(* IEC 61131-3 sources: std_i2980_v2.06_cp053/Source/IMM/ieccontrol/PumpGeneral (part 2) *)

(* ---- ABPumpOutput.pu ---- *)
(*
@h    ! WARNING !
@h    The Kemro K2 system (including software) only meets category B according to EN 954-1,
@h    thus it is not intended for usage in safety-relevant control applications in the field
@h    of personal safety (e.g. emergency stop).
@h    To implement potentially necessary safety-relevant control tasks, always use additional
@h    external safety devices that are intended for the particular purpose, and meet the necessary
@h    functional safety.
@h    For further information see EN 954-1 (EN ISO 13849-1) and/or the K2-x00 user manual, chapter
@h    "CE conformity, directives and standards".

This AB starts and stopps the process algorithms for fast output and mid output.
After a change in pressure or velocity lintab, a minimum output voltage is calculated.
During operation modes manual, HA and FA the output to the pump is at least this calculated minimum voltage,
even if there is actually no movement active.
In setup mode, the output voltage is set to 0.0 if the pump is stopped.
This block offers also the possibility to add a dither signal to pressure and velocity output.
Setting the dither amplitude to 0.0 disables the signal.
If the application is not running on a CP 03x, the dither amplitude is automatically resetted to 0.0.
*)

IMPORT_OVER_LISTFILE
 SET_ALARM
, GET_SYNC_REFTO
, WRITE_SVREAL_DIRECT
, FAddToScopeGroup
, ABAnalogOutput
, ABAnalogHWOut
, tsDeviceId
, KAPPL_LintabData
, tnOperationMode
, tnAnaOutputMode
, FBDebugTrace
, FBSinus
, KSWO_Status
, KCTRL_Lintab_Light
, KCTRL_Lintab_Param_Light
, KCAT_HandleData
, KCAT_Status

END_IMPORT

ALGORITHM_BLOCK ABPumpOutput #DUMMY_EDIT_BLOCK

SYSTEM_VAR
 sv_rPressure : REAL;
 sv_rVelocity : REAL;
 sv_DeviceId : tsDeviceId;
 sv_rMinVoltageVelOutput : REAL;
 sv_rMinVoltagePressOutput : REAL;
 sv_VelocityLintab : KAPPL_LintabData;
 sv_PressureLintab : KAPPL_LintabData;
 sv_OperationMode : tnOperationMode;
 sv_rValueMinVoltageVelDetect : REAL (* x - value [%] for detection of minimum output voltage of AO pump velocity *);
 sv_rValueMinVoltagePresDetect : REAL (* x - value [bar] for detection of minimum output voltage of AO pump pressure *);
 sv_rDitherFrequencyVel : REAL;
 sv_rDitherAmplitudeVel : REAL;
 sv_rDitherFrequencyPres : REAL;
 sv_rDitherAmplitudePres : REAL;
 sv_bInitStart : BOOL;
 sv_bInitDone : BOOL;
 sv_rMaxPressure : REAL;
END_VAR

SYSTEM_OBJECT
 TaskAnalog : TASK;
 TaskInject : TASK;
 TaskSlow : TASK;
 erVariableNotLinked : ALARM;
 PU_Task_7 : TASK;
 PU_Task_3 : TASK;
END_OBJECT

VAR
 mbStop : BOOL;
 mbStopped : BOOL := TRUE;
 mprPressureSource : REFTO REAL;
 mprVelocitySource : REFTO REAL;
 abAnalogOutputP : ABAnalogOutput;
 abAnalogOutputV : ABAnalogOutput;
 abAnalogHWOutP : ABAnalogHWOut;
 abAnalogHWOutV : ABAnalogHWOut;
 mrMinVoltageVelocityOutput : REAL (* minimum voltage for AO velocity (only considered in HA and FA) *);
 mrMinVoltagePressureOutput : REAL (* minimum voltage for AO pressure (only considered in HA and FA) *);
END_VAR

ALGORITHM aStart

VAR_INPUT
 AnaOutMode : tnAnaOutputMode;
 pLintabP : REFTO KAPPL_LintabData;
 pLintabV : REFTO KAPPL_LintabData;
 prPressure : REFTO REAL;
 prVelocity : REFTO REAL;
END_VAR
#BEGIN_EDIT_BLOCK
(**************************************** WARNING ********************************************
 *** The KEBA Kemro K2 System including software is not intended for safety control tasks! ***
 ***                       For further information see Comment tab!                        ***
 *********************************************************************************************)

mbStop := FALSE;
//make sure when we get a start and a stop very fast,
//we do not end up in a situation where mbStopped is FALSE but paXxxOutput is still running
mbStopped := FALSE;

abAnalogOutputP.aInit(pLintab := pLintabP);
abAnalogOutputV.aInit(pLintab := pLintabV);

mprPressureSource := prPressure;
mprVelocitySource := prVelocity;

CASE AnaOutMode OF

   nAnaOutputModeMid:
         START_PROCESS_ALGORITHM(paMidOutput);

   nAnaOutputModeFast:
         START_PROCESS_ALGORITHM(paFastOutput);
END_CASE;

;#END_EDIT_BLOCK END_ALGORITHM

ALGORITHM aStop

VAR_OUTPUT
 bReady : BOOL;
END_VAR
#BEGIN_EDIT_BLOCK
(**************************************** WARNING ********************************************
 *** The KEBA Kemro K2 System including software is not intended for safety control tasks! ***
 ***                       For further information see Comment tab!                        ***
 *********************************************************************************************)

IF NOT mbStopped THEN
   mbStop := TRUE;
END_IF;
bReady := mbStopped;

;#END_EDIT_BLOCK END_ALGORITHM

ALGORITHM aSetErrorMessage

VAR
 fbDebugTrace : FBDebugTrace;
END_VAR
#BEGIN_EDIT_BLOCK
(**************************************** WARNING ********************************************
 *** The KEBA Kemro K2 System including software is not intended for safety control tasks! ***
 ***                       For further information see Comment tab!                        ***
 *********************************************************************************************)

IF NOT abAnalogHWOutV.aIsLinked() THEN
   SET_ALARM(Name := erVariableNotLinked,
             SubID1 := sv_DeviceId.CompId,
             SubID2 := sv_DeviceId.IndexId,
             Param1 := 'ao_Velocity');
END_IF;

IF NOT abAnalogHWOutP.aIsLinked() THEN
   SET_ALARM(Name := erVariableNotLinked,
             SubID1 := sv_DeviceId.CompId,
             SubID2 := sv_DeviceId.IndexId,
             Param1 := 'ao_Pressure');
END_IF;

IF abAnalogOutputP.aRun.bError THEN
   fbDebugTrace(CONCAT('ABPumpOutput: error ',DINT_TO_STRING(abAnalogOutputP.aRun.iErrorInfo),' in ABAnalogOutputP'));
END_IF;

IF abAnalogOutputV.aRun.bError THEN
   fbDebugTrace(CONCAT('ABPumpOutput: error ',DINT_TO_STRING(abAnalogOutputV.aRun.iErrorInfo),' in ABAnalogOutputV'));
END_IF;

;#END_EDIT_BLOCK END_ALGORITHM

PROCESS_ALGORITHM paFastOutput ON TaskInject(15000)

VAR_TEMP
 b : BOOL;
END_VAR

VAR
 fbSinusVel : FBSinus;
 fbSinusPres : FBSinus;
 rDitherVel : REAL;
 rDitherPres : REAL;
 rPressure : REAL;
END_VAR

(* IecGraph-Code *)

(* init step *)
INITIAL_STEP OUT:
Init (P);
ADitherSignal (N);
AOUT (N);
END_STEP

ACTION Init: #BEGIN_EDIT_BLOCK
mbStopped := FALSE;

;#END_EDIT_BLOCK END_ACTION (*Init*)
ACTION AOUT: #BEGIN_EDIT_BLOCK
//limit pressure output to max. pressure of the pump
rPressure := MIN(sv_rMaxPressure, mprPressureSource^);

b := WRITE_SVREAL_DIRECT(sv_rPressure, rPressure);
b := WRITE_SVREAL_DIRECT(sv_rVelocity, mprVelocitySource^);

(* Lintab Calculation *)
abAnalogOutputP.aRun(rSetValue := sv_rPressure);
abAnalogOutputV.aRun(rSetValue := sv_rVelocity);

(* Output to AO and Shortcircuit detection *)
abAnalogHWOutP.aOut(rValue := (MAX(abAnalogOutputP.aRun.rOutput, mrMinVoltagePressureOutput)) + rDitherPres);
abAnalogHWOutV.aOut(rValue := (MAX(abAnalogOutputV.aRun.rOutput, mrMinVoltageVelocityOutput)) + rDitherVel);

;#END_EDIT_BLOCK END_ACTION (*AOUT*)

(* steps *)
STEP ERROR_STOP:
AErrorStop (P);
END_STEP

ACTION AErrorStop: #BEGIN_EDIT_BLOCK
sv_rPressure := 0.0;
sv_rVelocity := 0.0;
aSetErrorMessage();

;#END_EDIT_BLOCK END_ACTION (*AErrorStop*)
STEP S_Stop:
AStop (P);
END_STEP

ACTION AStop: #BEGIN_EDIT_BLOCK
mbStop := FALSE;

(* Stopping Analog Output*)
abAnalogHWOutP.aOut(rValue := mrMinVoltagePressureOutput);
abAnalogHWOutV.aOut(rValue := mrMinVoltageVelocityOutput);

mbStopped := TRUE;
STOP_PROCESS_ALGORITHM();

;#END_EDIT_BLOCK END_ACTION (*AStop*)

(* transitions *)
TRANSITION Trans1 (* Trans1 *) FROM OUT TO ERROR_STOP :=  #BEGIN_EDIT_BLOCK
abAnalogOutputP.aRun.bError OR
abAnalogOutputV.aRun.bError OR
abAnalogHWOutP.aOut.bError OR
abAnalogHWOutV.aOut.bError
;#END_EDIT_BLOCK
END_TRANSITION

GO_ON_TRANSITION Trans5 (* Trans5 *) FROM ERROR_STOP TO S_Stop :=  #BEGIN_EDIT_BLOCK
TRUE
;#END_EDIT_BLOCK
END_TRANSITION

GO_ON_TRANSITION TStop (* Trans4 *) FROM OUT TO S_Stop :=  #BEGIN_EDIT_BLOCK
mbStop
;#END_EDIT_BLOCK
END_TRANSITION

TRANSITION TNewOutput (* Trans7 *) FROM S_Stop TO OUT :=  #BEGIN_EDIT_BLOCK
TRUE
;#END_EDIT_BLOCK
END_TRANSITION

(* end IecGraph-Code *)
(* sfc-code *)

(* stand alone actions *)
ACTION ADitherSignal: #BEGIN_EDIT_BLOCK
(**************************************** WARNING ********************************************
 *** The KEBA Kemro K2 System including software is not intended for safety control tasks! ***
 ***                       For further information see Comment tab!                        ***
 *********************************************************************************************)

//sinus signals for pressure and velocity dither
IF sv_rDitherAmplitudeVel > 0.0 THEN
   fbSinusVel(rAmplitude := sv_rDitherAmplitudeVel,
              rFrequency := sv_rDitherFrequencyVel,
              rOut => rDitherVel);
ELSE
   rDitherVel := 0.0;
END_IF;

IF sv_rDitherAmplitudePres > 0.0 THEN
   fbSinusPres(rAmplitude := sv_rDitherAmplitudePres,
              rFrequency := sv_rDitherFrequencyPres,
              rOut => rDitherPres);
ELSE
   rDitherPres := 0.0;
END_IF;

;#END_EDIT_BLOCK END_ACTION (*ADitherSignal*)
(* end sfc-code *)

END_ALGORITHM

PROCESS_ALGORITHM paMidOutput ON TaskAnalog(15000)

VAR_TEMP
 b : BOOL;
END_VAR

VAR
 fbSinusVel : FBSinus;
 fbSinusPres : FBSinus;
 rDitherVel : REAL;
 rDitherPres : REAL;
 rPressure : REAL;
END_VAR

(* IecGraph-Code *)

(* init step *)
INITIAL_STEP OUT:
Init (P);
ADitherSignal (N);
AOUT (N);
END_STEP

ACTION Init: #BEGIN_EDIT_BLOCK
mbStopped := FALSE;

;#END_EDIT_BLOCK END_ACTION (*Init*)
ACTION AOUT: #BEGIN_EDIT_BLOCK
//limit pressure output to max. pressure of the pump
rPressure := MIN(sv_rMaxPressure, mprPressureSource^);

b := WRITE_SVREAL_DIRECT(sv_rPressure, rPressure);
b := WRITE_SVREAL_DIRECT(sv_rVelocity, mprVelocitySource^);

(* Lintab Calculation *)
abAnalogOutputP.aRun(rSetValue := sv_rPressure);
abAnalogOutputV.aRun(rSetValue := sv_rVelocity);

(* Shortcircuit detection *)
abAnalogHWOutP.aOut(rValue := (MAX(abAnalogOutputP.aRun.rOutput, mrMinVoltagePressureOutput)) + rDitherPres);
abAnalogHWOutV.aOut(rValue := (MAX(abAnalogOutputV.aRun.rOutput, mrMinVoltageVelocityOutput)) + rDitherVel);

;#END_EDIT_BLOCK END_ACTION (*AOUT*)

(* steps *)
STEP ERROR_STOP:
AErrorStop (P);
END_STEP

ACTION AErrorStop: #BEGIN_EDIT_BLOCK
sv_rPressure := 0.0;
sv_rVelocity := 0.0;
aSetErrorMessage();

;#END_EDIT_BLOCK END_ACTION (*AErrorStop*)
STEP S_Stop:
AStop (P);
END_STEP

ACTION AStop: #BEGIN_EDIT_BLOCK
mbStop := FALSE;

(* Stopping Analog Output*)
abAnalogHWOutP.aOut(rValue := mrMinVoltagePressureOutput);
abAnalogHWOutV.aOut(rValue := mrMinVoltageVelocityOutput);

mbStopped := TRUE;
STOP_PROCESS_ALGORITHM();

;#END_EDIT_BLOCK END_ACTION (*AStop*)

(* transitions *)
TRANSITION Trans1 (* Trans1 *) FROM OUT TO ERROR_STOP :=  #BEGIN_EDIT_BLOCK
abAnalogOutputP.aRun.bError OR
abAnalogOutputV.aRun.bError OR
abAnalogHWOutP.aOut.bError OR
abAnalogHWOutV.aOut.bError
;#END_EDIT_BLOCK
END_TRANSITION

GO_ON_TRANSITION Trans5 (* Trans5 *) FROM ERROR_STOP TO S_Stop :=  #BEGIN_EDIT_BLOCK
TRUE
;#END_EDIT_BLOCK
END_TRANSITION

GO_ON_TRANSITION TStop (* Trans4 *) FROM OUT TO S_Stop :=  #BEGIN_EDIT_BLOCK
mbStop
;#END_EDIT_BLOCK
END_TRANSITION

TRANSITION TNewOutput (* Trans7 *) FROM S_Stop TO OUT :=  #BEGIN_EDIT_BLOCK
TRUE
;#END_EDIT_BLOCK
END_TRANSITION

(* end IecGraph-Code *)
(* sfc-code *)

(* stand alone actions *)
ACTION ADitherSignal: #BEGIN_EDIT_BLOCK
(**************************************** WARNING ********************************************
 *** The KEBA Kemro K2 System including software is not intended for safety control tasks! ***
 ***                       For further information see Comment tab!                        ***
 *********************************************************************************************)

//sinus signals for pressure and velocity dither
IF sv_rDitherAmplitudeVel > 0.0 THEN
   fbSinusVel(rAmplitude := sv_rDitherAmplitudeVel,
              rFrequency := sv_rDitherFrequencyVel,
              rOut => rDitherVel);
ELSE
   rDitherVel := 0.0;
END_IF;

IF sv_rDitherAmplitudePres > 0.0 THEN
   fbSinusPres(rAmplitude := sv_rDitherAmplitudePres,
              rFrequency := sv_rDitherFrequencyPres,
              rOut => rDitherPres);
ELSE
   rDitherPres := 0.0;
END_IF;

;#END_EDIT_BLOCK END_ACTION (*ADitherSignal*)
(* end sfc-code *)

END_ALGORITHM

PROCESS_ALGORITHM paInitDebugMeasurement ON TaskSlow AUTOSTART

VAR
 fuName : STRING(255);
 variableName : STRING(255);
 swoState : KSWO_Status;
 b : BOOL;
END_VAR
#BEGIN_EDIT_BLOCK
fuName := GET_MY_FU_NAME();
variableName := CONCAT(fuName,'.rPressure Hydr bar');
swoState := KSWO_AddVariable( Task := TaskInject,
                              Name := variableName,
                              Variable := sv_rPressure);
b := FAddToScopeGroup(Task := TaskInject,
                      Name := variableName,
                      GroupId := cScopeGroupPump);
variableName := CONCAT(fuName,'.rVelocity %');
swoState := KSWO_AddVariable( Task := TaskInject,
                              Name := variableName,
                              Variable := sv_rVelocity);
b := FAddToScopeGroup(Task := TaskInject,
                      Name := variableName,
                      GroupId := cScopeGroupPump);

variableName := CONCAT(fuName,'.rPressure Hydr bar');
swoState := KSWO_AddVariable( Task := TaskAnalog,
                              Name := variableName,
                              Variable := sv_rPressure);
variableName := CONCAT(fuName,'.rVelocity %');
swoState := KSWO_AddVariable( Task := TaskAnalog,
                              Name := variableName,
                              Variable := sv_rVelocity);

STOP_PROCESS_ALGORITHM();

;#END_EDIT_BLOCK END_ALGORITHM

ALGORITHM aGetMinVoltage

VAR_INPUT
 pLintab : REFTO KAPPL_LintabData;
 rXValue : REAL (* xValue (for example 1% or 2 bar) *);
END_VAR

VAR_OUTPUT
 rMinVoltage : REAL (* according voltage for rXValue *);
END_VAR

VAR
 Lintab : KCTRL_Lintab_Light;
 LintabParams : KCTRL_Lintab_Param_Light;
END_VAR
#BEGIN_EDIT_BLOCK
(**************************************** WARNING ********************************************
 *** The KEBA Kemro K2 System including software is not intended for safety control tasks! ***
 ***                       For further information see Comment tab!                        ***
 *********************************************************************************************)

LintabParams.LintabPoints := pLintab^.LintabPoints;
LintabParams.Mode.bLinearExtrapolation := TRUE;
LintabParams.Mode.bSetNegativeValuesToZero := FALSE;
LintabParams.Mode.bZeroExtrapolation := FALSE;
Lintab.Par(Param := LintabParams);

IF Lintab.Par.parStatus <> KCTRL_Ret_OK THEN
   rMinVoltage := 0.0;
   RETURN; //error -> return 0.0
END_IF;

//calculate value
Lintab.Calculate(rX := rXValue);
IF Lintab.Calculate.calcStatus <> KCTRL_Ret_OK THEN
   rMinVoltage := 0.0;
   RETURN; //error -> return 0.0
ELSE
   rMinVoltage := Lintab.Calculate.rY;
END_IF;

;#END_EDIT_BLOCK END_ALGORITHM

POSTUPDATE_ALGORITHM pVelocityLintab ON PU_Task_7 WITH sv_VelocityLintab,sv_rValueMinVoltageVelDetect

#BEGIN_EDIT_BLOCK
(**************************************** WARNING ********************************************
 *** The KEBA Kemro K2 System including software is not intended for safety control tasks! ***
 ***                       For further information see Comment tab!                        ***
 *********************************************************************************************)

aGetMinVoltage(pLintab := @sv_VelocityLintab,
               rXValue := sv_rValueMinVoltageVelDetect,
               rMinVoltage => sv_rMinVoltageVelOutput);

;#END_EDIT_BLOCK END_ALGORITHM

POSTUPDATE_ALGORITHM pPressureLintab ON PU_Task_7 WITH sv_PressureLintab,sv_rValueMinVoltagePresDetect

#BEGIN_EDIT_BLOCK
(**************************************** WARNING ********************************************
 *** The KEBA Kemro K2 System including software is not intended for safety control tasks! ***
 ***                       For further information see Comment tab!                        ***
 *********************************************************************************************)

aGetMinVoltage(pLintab := @sv_PressureLintab,
               rXValue := sv_rValueMinVoltagePresDetect,
               rMinVoltage => sv_rMinVoltagePressOutput);

;#END_EDIT_BLOCK END_ALGORITHM

POSTUPDATE_ALGORITHM pDitherParams ON PU_Task_7 WITH sv_bInitStart,sv_rDitherAmplitudePres,sv_rDitherAmplitudeVel

VAR
 HandleData : KCAT_HandleData;
 CatStatus : KCAT_Status;
 sDevice : STRING(31);
 bInitDone : BOOL;
 bCurrentOutput : BOOL (* TRUE: current output available *);
END_VAR
#BEGIN_EDIT_BLOCK
(**************************************** WARNING ********************************************
 *** The KEBA Kemro K2 System including software is not intended for safety control tasks! ***
 ***                       For further information see Comment tab!                        ***
 *********************************************************************************************)

IF NOT bInitDone THEN
   //get device name
   HandleData := KCAT_GetHandle('IO.ONBOARD.deviceName');
   IF HandleData.Status = KCAT_Status_OK THEN
      CatStatus := KCAT_GetValue(Handle := HandleData.Handle, Buffer := sDevice);
      sDevice := LEFT(sDevice,5);

      IF sDevice ='CP 03' THEN
         bCurrentOutput := TRUE;
      END_IF;
   END_IF;

   bInitDone := TRUE;

END_IF;

IF NOT bCurrentOutput THEN
   //set dither amplitude to 0.0 (=disable dither signal)
   sv_rDitherAmplitudeVel := 0.0;
   sv_rDitherAmplitudePres := 0.0;
END_IF;

;#END_EDIT_BLOCK END_ALGORITHM

POSTUPDATE_ALGORITHM pSetMinVoltage ON PU_Task_3 WITH sv_bInitDone,sv_rMinVoltageVelOutput,sv_rMinVoltagePressOutput,sv_OperationMode

#BEGIN_EDIT_BLOCK
(**************************************** WARNING ********************************************
 *** The KEBA Kemro K2 System including software is not intended for safety control tasks! ***
 ***                       For further information see Comment tab!                        ***
 *********************************************************************************************)

IF sv_OperationMode = nSetup THEN
   //setup mode -> set minimum output voltage to 0.0
   mrMinVoltagePressureOutput := 0.0;
   mrMinVoltageVelocityOutput := 0.0;

ELSE
   //all other operation modes
   mrMinVoltagePressureOutput := sv_rMinVoltagePressOutput;
   mrMinVoltageVelocityOutput := sv_rMinVoltageVelOutput;
END_IF;

IF mbStopped THEN
   //write to AO´s immediately if device is not active
   abAnalogHWOutP.aOut(rValue := mrMinVoltagePressureOutput);
   abAnalogHWOutV.aOut(rValue := mrMinVoltageVelocityOutput);
END_IF;

;#END_EDIT_BLOCK END_ALGORITHM

END_ALGORITHM_BLOCK

#END_OF_IEC_PART

@Puma @IecEditor 6 97 @Pou 25
@@@BEG_Comment@@@
@h    ! WARNING !
@h    The Kemro K2 system (including software) only meets category B according to EN 954-1,
@h    thus it is not intended for usage in safety-relevant control applications in the field
@h    of personal safety (e.g. emergency stop).
@h    To implement potentially necessary safety-relevant control tasks, always use additional
@h    external safety devices that are intended for the particular purpose, and meet the necessary
@h    functional safety.
@h    For further information see EN 954-1 (EN ISO 13849-1) and/or the K2-x00 user manual, chapter
@h    "CE conformity, directives and standards".

This AB starts and stopps the process algorithms for fast output and mid output.
After a change in pressure or velocity lintab, a minimum output voltage is calculated.
During operation modes manual, HA and FA the output to the pump is at least this calculated minimum voltage,
even if there is actually no movement active.
In setup mode, the output voltage is set to 0.0 if the pump is stopped.
This block offers also the possibility to add a dither signal to pressure and velocity output.
Setting the dither amplitude to 0.0 disables the signal.
If the application is not running on a CP 03x, the dither amplitude is automatically resetted to 0.0.
@@@END_Comment@@@

@BEG_Contents

@BEG_Func
@RT(17)FuncTreeContainer
4
@Var @RT(9)SET_ALARM @RT(0) @T @T @DERIVED 0 @F @RT(23)KEBA_STANDARD_PROCEDURE @F
@T
@BEG_Attrib
0 @RT(0) @RT(0)
@END_Attrib
1 1 @F @F @F @F

@Var @RT(14)GET_SYNC_REFTO @RT(0) @T @T @DERIVED 0 @F @RT(22)KEBA_STANDARD_FUNCTION @F
@T
@BEG_Attrib
0 @RT(0) @RT(0)
@END_Attrib
1 1 @F @F @F @F

@Var @RT(19)WRITE_SVREAL_DIRECT @RT(0) @T @T @DERIVED 0 @F @RT(22)KEBA_STANDARD_FUNCTION @F
@T
@BEG_Attrib
0 @RT(0) @RT(0)
@END_Attrib
1 1 @F @F @F @F

@Var @RT(16)FAddToScopeGroup @RT(0) @T @T @DERIVED 0 @F @RT(8)FUNCTION @F
@T
@BEG_Attrib
0 @RT(0) @RT(0)
@END_Attrib
1 1 @F @F @F @F

@END_Func

@BEG_Const
@RT(18)ConstTreeContainer
0
@END_Const

@BEG_Export

@BEG_Kind
@ALGORITHM_BLOCK @RT(12)ABPumpOutput @STRUCTURED_TEXT
@RT(0) @RT(0) @RT(0)
@END_Kind

@BEG_Dcl
@RT(16)DclTreeContainer
33
@Var @RT(10)TaskAnalog @RT(0) @T @T @RENAMED 0 @T @T @DT @RT(4)TASK @RT(0) @T @T @BASIC 0 @F
@F @F
@T
@BEG_Attrib
3 @RT(0) @RT(0) @RT(0)
@END_Attrib
1 7 @F @F @F @F

@Var @RT(10)TaskInject @RT(0) @T @T @RENAMED 0 @T @T @DT @RT(4)TASK @RT(0) @T @T @BASIC 0 @F
@F @F
@T
@BEG_Attrib
3 @RT(0) @RT(0) @RT(0)
@END_Attrib
1 7 @F @F @F @F

@Var @RT(8)TaskSlow @RT(0) @T @T @RENAMED 0 @T @T @DT @RT(4)TASK @RT(0) @T @T @BASIC 0 @F
@F @F
@T
@BEG_Attrib
3 @RT(0) @RT(0) @RT(0)
@END_Attrib
1 7 @F @F @F @F

@Var @RT(12)sv_rPressure @RT(0) @T @F @DT @RT(4)REAL @RT(0) @T @T @BASIC 0 @F
@F @F
@T
@BEG_Attrib
3 @RT(0) @RT(0) @RT(0)
@END_Attrib
1 8 @F @F @F @F

@Var @RT(12)sv_rVelocity @RT(0) @T @F @DT @RT(4)REAL @RT(0) @T @T @BASIC 0 @F
@F @F
@T
@BEG_Attrib
3 @RT(0) @RT(0) @RT(0)
@END_Attrib
1 8 @F @F @F @F

@Var @RT(6)mbStop @RT(0) @T @F @DT @RT(4)BOOL @RT(0) @T @T @BASIC 0 @F
@F @F
@T
@BEG_Attrib
3 @RT(0) @RT(0) @RT(0)
@END_Attrib
1 0 @F @F @F @F

@Var @RT(9)mbStopped @RT(0) @T @F @DT @RT(4)BOOL @RT(0) @T @T @BASIC 0 @F
@F @F
@T
@BEG_Attrib
3 @RT(4)TRUE @RT(0) @RT(0)
@END_Attrib
1 0 @F @F @F @F

@Var @RT(17)mprPressureSource @RT(0) @T @T @REFTO 0 @T @DT @RT(4)REAL @RT(0) @T @T @BASIC 0 @F
@F @F
@T
@BEG_Attrib
3 @RT(0) @RT(0) @RT(0)
@END_Attrib
1 0 @F @F @F @F

@Var @RT(17)mprVelocitySource @RT(0) @T @T @REFTO 0 @T @DT @RT(4)REAL @RT(0) @T @T @BASIC 0 @F
@F @F
@T
@BEG_Attrib
3 @RT(0) @RT(0) @RT(0)
@END_Attrib
1 0 @F @F @F @F

@Var @RT(15)abAnalogOutputP @RT(0) @T @T @DERIVED 0 @T @T @DT @RT(14)ABAnalogOutput @RT(0) @T @T @UNKNOWN 0 @F
@F @F
@T
@BEG_Attrib
3 @RT(0) @RT(0) @RT(0)
@END_Attrib
1 0 @F @F @F @F

@Var @RT(15)abAnalogOutputV @RT(0) @T @T @DERIVED 0 @T @T @DT @RT(14)ABAnalogOutput @RT(0) @T @T @UNKNOWN 0 @F
@F @F
@T
@BEG_Attrib
3 @RT(0) @RT(0) @RT(0)
@END_Attrib
1 0 @F @F @F @F

@Var @RT(14)abAnalogHWOutP @RT(0) @T @T @DERIVED 0 @T @T @DT @RT(13)ABAnalogHWOut @RT(0) @T @T @UNKNOWN 0 @F
@F @F
@T
@BEG_Attrib
3 @RT(0) @RT(0) @RT(0)
@END_Attrib
1 0 @F @F @F @F

@Var @RT(14)abAnalogHWOutV @RT(0) @T @T @DERIVED 0 @T @T @DT @RT(13)ABAnalogHWOut @RT(0) @T @T @UNKNOWN 0 @F
@F @F
@T
@BEG_Attrib
3 @RT(0) @RT(0) @RT(0)
@END_Attrib
1 0 @F @F @F @F

@Var @RT(19)erVariableNotLinked @RT(0) @T @F @DT @RT(5)ALARM @RT(0) @T @T @BASIC 0 @F
@F @F
@T
@BEG_Attrib
3 @RT(0) @RT(0) @RT(0)
@END_Attrib
1 7 @F @F @F @F

@Var @RT(11)sv_DeviceId @RT(0) @T @T @DERIVED 0 @T @T @DT @RT(10)tsDeviceId @RT(0) @T @T @UNKNOWN 0 @F
@F @F
@T
@BEG_Attrib
3 @RT(0) @RT(0) @RT(0)
@END_Attrib
1 8 @F @F @F @F

@Var @RT(23)sv_rMinVoltageVelOutput @RT(0) @T @F @DT @RT(4)REAL @RT(0) @T @T @BASIC 0 @F
@F @F
@T
@BEG_Attrib
3 @RT(0) @RT(0) @RT(0)
@END_Attrib
1 8 @F @F @F @F

@Var @RT(25)sv_rMinVoltagePressOutput @RT(0) @T @F @DT @RT(4)REAL @RT(0) @T @T @BASIC 0 @F
@F @F
@T
@BEG_Attrib
3 @RT(0) @RT(0) @RT(0)
@END_Attrib
1 8 @F @F @F @F

@Var @RT(9)PU_Task_7 @RT(0) @T @T @RENAMED 0 @T @T @DT @RT(4)TASK @RT(0) @T @T @BASIC 0 @F
@F @F
@T
@BEG_Attrib
3 @RT(0) @RT(0) @RT(0)
@END_Attrib
1 7 @F @F @F @F

@Var @RT(9)PU_Task_3 @RT(0) @T @T @RENAMED 0 @T @T @DT @RT(4)TASK @RT(0) @T @T @BASIC 0 @F
@F @F
@T
@BEG_Attrib
3 @RT(0) @RT(0) @RT(0)
@END_Attrib
1 7 @F @F @F @F

@Var @RT(17)sv_VelocityLintab @RT(0) @T @T @DERIVED 0 @T @T @DT @RT(16)KAPPL_LintabData @RT(0) @T @T @UNKNOWN 0 @F
@F @F
@T
@BEG_Attrib
3 @RT(0) @RT(0) @RT(0)
@END_Attrib
1 8 @F @F @F @F

@Var @RT(17)sv_PressureLintab @RT(0) @T @T @DERIVED 0 @T @T @DT @RT(16)KAPPL_LintabData @RT(0) @T @T @UNKNOWN 0 @F
@F @F
@T
@BEG_Attrib
3 @RT(0) @RT(0) @RT(0)
@END_Attrib
1 8 @F @F @F @F

@Var @RT(16)sv_OperationMode @RT(0) @T @T @DERIVED 0 @T @T @DT @RT(15)tnOperationMode @RT(0) @T @T @UNKNOWN 0 @F
@F @F
@T
@BEG_Attrib
3 @RT(0) @RT(0) @RT(0)
@END_Attrib
1 8 @F @F @F @F

@Var @RT(26)mrMinVoltageVelocityOutput @RT(0) @T @F @DT @RT(4)REAL @RT(0) @T @T @BASIC 0 @F
@F @F
@T
@BEG_Attrib
3 @RT(0) @RT(62)minimum voltage for AO velocity (only considered in HA and FA) @RT(0)
@END_Attrib
1 0 @F @F @F @F

@Var @RT(26)mrMinVoltagePressureOutput @RT(0) @T @F @DT @RT(4)REAL @RT(0) @T @T @BASIC 0 @F
@F @F
@T
@BEG_Attrib
3 @RT(0) @RT(62)minimum voltage for AO pressure (only considered in HA and FA) @RT(0)
@END_Attrib
1 0 @F @F @F @F

@Var @RT(28)sv_rValueMinVoltageVelDetect @RT(0) @T @F @DT @RT(4)REAL @RT(0) @T @T @BASIC 0 @F
@F @F
@T
@BEG_Attrib
3 @RT(0) @RT(73)x - value [%] for detection of minimum output voltage of AO pump velocity @RT(0)
@END_Attrib
1 8 @F @F @F @F

@Var @RT(29)sv_rValueMinVoltagePresDetect @RT(0) @T @F @DT @RT(4)REAL @RT(0) @T @T @BASIC 0 @F
@F @F
@T
@BEG_Attrib
3 @RT(0) @RT(75)x - value [bar] for detection of minimum output voltage of AO pump pressure @RT(0)
@END_Attrib
1 8 @F @F @F @F

@Var @RT(22)sv_rDitherFrequencyVel @RT(0) @T @F @DT @RT(4)REAL @RT(0) @T @T @BASIC 0 @F
@F @F
@T
@BEG_Attrib
3 @RT(0) @RT(0) @RT(0)
@END_Attrib
1 8 @F @F @F @F

@Var @RT(22)sv_rDitherAmplitudeVel @RT(0) @T @F @DT @RT(4)REAL @RT(0) @T @T @BASIC 0 @F
@F @F
@T
@BEG_Attrib
3 @RT(0) @RT(0) @RT(0)
@END_Attrib
1 8 @F @F @F @F

@Var @RT(23)sv_rDitherFrequencyPres @RT(0) @T @F @DT @RT(4)REAL @RT(0) @T @T @BASIC 0 @F
@F @F
@T
@BEG_Attrib
3 @RT(0) @RT(0) @RT(0)
@END_Attrib
1 8 @F @F @F @F

@Var @RT(23)sv_rDitherAmplitudePres @RT(0) @T @F @DT @RT(4)REAL @RT(0) @T @T @BASIC 0 @F
@F @F
@T
@BEG_Attrib
3 @RT(0) @RT(0) @RT(0)
@END_Attrib
1 8 @F @F @F @F

@Var @RT(13)sv_bInitStart @RT(0) @T @T @RENAMED 0 @T @T @DT @RT(4)BOOL @RT(0) @T @T @BASIC 0 @F
@F @F
@T
@BEG_Attrib
3 @RT(0) @RT(0) @RT(0)
@END_Attrib
1 8 @F @F @F @F

@Var @RT(12)sv_bInitDone @RT(0) @T @F @DT @RT(4)BOOL @RT(0) @T @T @BASIC 0 @F
@F @F
@T
@BEG_Attrib
3 @RT(0) @RT(0) @RT(0)
@END_Attrib
1 8 @F @F @F @F

@Var @RT(15)sv_rMaxPressure @RT(0) @T @F @DT @RT(4)REAL @RT(0) @T @T @BASIC 0 @F
@F @F
@T
@BEG_Attrib
3 @RT(0) @RT(0) @RT(0)
@END_Attrib
1 8 @F @F @F @F

@END_Dcl

@END_Export

@BEG_Body

11

@BEG_Export

@BEG_Algo
@ALGORITHM @RT(6)aStart @STRUCTURED_TEXT
@RT(0) @RT(0) @RT(0) @F @F
@END_Algo

@BEG_Dcl
@RT(16)DclTreeContainer
5
@Var @RT(10)AnaOutMode @RT(0) @T @T @DERIVED 0 @T @T @DT @RT(15)tnAnaOutputMode @RT(0) @T @T @UNKNOWN 0 @F
@F @F
@T
@BEG_Attrib
3 @RT(0) @RT(0) @RT(0)
@END_Attrib
1 1 @F @F @F @F

@Var @RT(8)pLintabP @RT(0) @T @T @REFTO 0 @F @DERIVED 0 @T @T @DT @RT(16)KAPPL_LintabData @RT(0) @T @T @UNKNOWN 0 @F
@F @F
@T
@BEG_Attrib
3 @RT(0) @RT(0) @RT(0)
@END_Attrib
1 1 @F @F @F @F

@Var @RT(8)pLintabV @RT(0) @T @T @REFTO 0 @F @DERIVED 0 @T @T @DT @RT(16)KAPPL_LintabData @RT(0) @T @T @UNKNOWN 0 @F
@F @F
@T
@BEG_Attrib
3 @RT(0) @RT(0) @RT(0)
@END_Attrib
1 1 @F @F @F @F

@Var @RT(10)prPressure @RT(0) @T @T @REFTO 0 @T @DT @RT(4)REAL @RT(0) @T @T @BASIC 0 @F
@F @F
@T
@BEG_Attrib
3 @RT(0) @RT(0) @RT(0)
@END_Attrib
1 1 @F @F @F @F

@Var @RT(10)prVelocity @RT(0) @T @T @REFTO 0 @T @DT @RT(4)REAL @RT(0) @T @T @BASIC 0 @F
@F @F
@T
@BEG_Attrib
3 @RT(0) @RT(0) @RT(0)
@END_Attrib
1 1 @F @F @F @F

@END_Dcl

@END_Export

@BEG_Export

@BEG_Algo
@ALGORITHM @RT(5)aStop @STRUCTURED_TEXT
@RT(0) @RT(0) @RT(0) @F @F
@END_Algo

@BEG_Dcl
@RT(16)DclTreeContainer
1
@Var @RT(6)bReady @RT(0) @T @F @DT @RT(4)BOOL @RT(0) @T @T @BASIC 0 @F
@F @F
@T
@BEG_Attrib
3 @RT(0) @RT(0) @RT(0)
@END_Attrib
1 3 @F @F @F @F

@END_Dcl

@END_Export

@BEG_Export

@BEG_Algo
@ALGORITHM @RT(16)aSetErrorMessage @STRUCTURED_TEXT
@RT(0) @RT(0) @RT(0) @F @F
@END_Algo

@BEG_Dcl
@RT(16)DclTreeContainer
1
@Var @RT(12)fbDebugTrace @RT(0) @T @T @DERIVED 0 @T @T @DT @RT(12)FBDebugTrace @RT(0) @T @T @UNKNOWN 0 @F
@F @F
@T
@BEG_Attrib
3 @RT(0) @RT(0) @RT(0)
@END_Attrib
1 0 @F @F @F @F

@END_Dcl

@END_Export

@BEG_Export

@BEG_Algo
@PROCESS_ALGORITHM @RT(12)paFastOutput @SEQUENTIAL_FLOW_CHART
@RT(0) @RT(0) @RT(17)TaskInject(15000) @F @F
@END_Algo

@BEG_Dcl
@RT(16)DclTreeContainer
6
@Var @RT(10)fbSinusVel @RT(0) @T @T @DERIVED 0 @T @T @DT @RT(7)FBSinus @RT(0) @T @T @UNKNOWN 0 @F
@F @F
@T
@BEG_Attrib
3 @RT(0) @RT(0) @RT(0)
@END_Attrib
1 0 @F @F @F @F

@Var @RT(11)fbSinusPres @RT(0) @T @T @DERIVED 0 @T @T @DT @RT(7)FBSinus @RT(0) @T @T @UNKNOWN 0 @F
@F @F
@T
@BEG_Attrib
3 @RT(0) @RT(0) @RT(0)
@END_Attrib
1 0 @F @F @F @F

@Var @RT(10)rDitherVel @RT(0) @T @F @DT @RT(4)REAL @RT(0) @T @T @BASIC 0 @F
@F @F
@T
@BEG_Attrib
3 @RT(0) @RT(0) @RT(0)
@END_Attrib
1 0 @F @F @F @F

@Var @RT(11)rDitherPres @RT(0) @T @F @DT @RT(4)REAL @RT(0) @T @T @BASIC 0 @F
@F @F
@T
@BEG_Attrib
3 @RT(0) @RT(0) @RT(0)
@END_Attrib
1 0 @F @F @F @F

@Var @RT(1)b @RT(0) @T @F @DT @RT(4)BOOL @RT(0) @T @T @BASIC 0 @F
@F @F
@T
@BEG_Attrib
3 @RT(0) @RT(0) @RT(0)
@END_Attrib
1 4 @F @F @F @F

@Var @RT(9)rPressure @RT(0) @T @F @DT @RT(4)REAL @RT(0) @T @T @BASIC 0 @F
@F @F
@T
@BEG_Attrib
3 @RT(0) @RT(0) @RT(0)
@END_Attrib
1 0 @F @F @F @F

@END_Dcl

@END_Export

@BEG_Export

@BEG_Algo
@PROCESS_ALGORITHM @RT(11)paMidOutput @SEQUENTIAL_FLOW_CHART
@RT(0) @RT(0) @RT(17)TaskAnalog(15000) @F @F
@END_Algo

@BEG_Dcl
@RT(16)DclTreeContainer
6
@Var @RT(10)fbSinusVel @RT(0) @T @T @DERIVED 0 @T @T @DT @RT(7)FBSinus @RT(0) @T @T @UNKNOWN 0 @F
@F @F
@T
@BEG_Attrib
3 @RT(0) @RT(0) @RT(0)
@END_Attrib
1 0 @F @F @F @F

@Var @RT(11)fbSinusPres @RT(0) @T @T @DERIVED 0 @T @T @DT @RT(7)FBSinus @RT(0) @T @T @UNKNOWN 0 @F
@F @F
@T
@BEG_Attrib
3 @RT(0) @RT(0) @RT(0)
@END_Attrib
1 0 @F @F @F @F

@Var @RT(10)rDitherVel @RT(0) @T @F @DT @RT(4)REAL @RT(0) @T @T @BASIC 0 @F
@F @F
@T
@BEG_Attrib
3 @RT(0) @RT(0) @RT(0)
@END_Attrib
1 0 @F @F @F @F

@Var @RT(11)rDitherPres @RT(0) @T @F @DT @RT(4)REAL @RT(0) @T @T @BASIC 0 @F
@F @F
@T
@BEG_Attrib
3 @RT(0) @RT(0) @RT(0)
@END_Attrib
1 0 @F @F @F @F

@Var @RT(1)b @RT(0) @T @F @DT @RT(4)BOOL @RT(0) @T @T @BASIC 0 @F
@F @F
@T
@BEG_Attrib
3 @RT(0) @RT(0) @RT(0)
@END_Attrib
1 4 @F @F @F @F

@Var @RT(9)rPressure @RT(0) @T @F @DT @RT(4)REAL @RT(0) @T @T @BASIC 0 @F
@F @F
@T
@BEG_Attrib
3 @RT(0) @RT(0) @RT(0)
@END_Attrib
1 0 @F @F @F @F

@END_Dcl

@END_Export

@BEG_Export

@BEG_Algo
@PROCESS_ALGORITHM @RT(22)paInitDebugMeasurement @STRUCTURED_TEXT
@RT(0) @RT(0) @RT(8)TaskSlow @T @F
@END_Algo

@BEG_Dcl
@RT(16)DclTreeContainer
4
@Var @RT(6)fuName @RT(0) @T @F @DT @RT(11)STRING(255) @RT(0) @T @T @STRING 0 @F @RT(3)255 @F
@F @F
@T
@BEG_Attrib
3 @RT(0) @RT(0) @RT(0)
@END_Attrib
1 0 @F @F @F @F

@Var @RT(12)variableName @RT(0) @T @F @DT @RT(11)STRING(255) @RT(0) @T @T @STRING 0 @F @RT(3)255 @F
@F @F
@T
@BEG_Attrib
3 @RT(0) @RT(0) @RT(0)
@END_Attrib
1 0 @F @F @F @F

@Var @RT(8)swoState @RT(0) @T @T @DERIVED 0 @T @T @DT @RT(11)KSWO_Status @RT(0) @T @T @UNKNOWN 0 @F
@F @F
@T
@BEG_Attrib
3 @RT(0) @RT(0) @RT(0)
@END_Attrib
1 0 @F @F @F @F

@Var @RT(1)b @RT(0) @T @F @DT @RT(4)BOOL @RT(0) @T @T @BASIC 0 @F
@F @F
@T
@BEG_Attrib
3 @RT(0) @RT(0) @RT(0)
@END_Attrib
1 0 @F @F @F @F

@END_Dcl

@END_Export

@BEG_Export

@BEG_Algo
@ALGORITHM @RT(14)aGetMinVoltage @STRUCTURED_TEXT
@RT(0) @RT(0) @RT(0) @F @F
@END_Algo

@BEG_Dcl
@RT(16)DclTreeContainer
5
@Var @RT(7)pLintab @RT(0) @T @T @REFTO 0 @F @DERIVED 0 @T @T @DT @RT(16)KAPPL_LintabData @RT(0) @T @T @UNKNOWN 0 @F
@F @F
@T
@BEG_Attrib
3 @RT(0) @RT(0) @RT(0)
@END_Attrib
1 1 @F @F @F @F

@Var @RT(7)rXValue @RT(0) @T @F @DT @RT(4)REAL @RT(0) @T @T @BASIC 0 @F
@F @F
@T
@BEG_Attrib
3 @RT(0) @RT(32)xValue (for example 1% or 2 bar) @RT(0)
@END_Attrib
1 1 @F @F @F @F

@Var @RT(11)rMinVoltage @RT(0) @T @F @DT @RT(4)REAL @RT(0) @T @T @BASIC 0 @F
@F @F
@T
@BEG_Attrib
3 @RT(0) @RT(29)according voltage for rXValue @RT(0)
@END_Attrib
1 3 @F @F @F @F

@Var @RT(6)Lintab @RT(0) @T @T @DERIVED 0 @T @T @DT @RT(18)KCTRL_Lintab_Light @RT(0) @T @T @UNKNOWN 0 @F
@F @F
@T
@BEG_Attrib
3 @RT(0) @RT(0) @RT(0)
@END_Attrib
1 0 @F @F @F @F

@Var @RT(12)LintabParams @RT(0) @T @T @DERIVED 0 @T @T @DT @RT(24)KCTRL_Lintab_Param_Light @RT(0) @T @T @UNKNOWN 0 @F
@F @F
@T
@BEG_Attrib
3 @RT(0) @RT(0) @RT(0)
@END_Attrib
1 0 @F @F @F @F

@END_Dcl

@END_Export

@BEG_Export

@BEG_Algo
@POSTUPDATE_ALGORITHM @RT(15)pVelocityLintab @STRUCTURED_TEXT
@RT(0) @RT(46)sv_VelocityLintab,sv_rValueMinVoltageVelDetect @RT(9)PU_Task_7 @F @F
@END_Algo

@BEG_Dcl
@RT(16)DclTreeContainer
0
@END_Dcl

@END_Export

@BEG_Export

@BEG_Algo
@POSTUPDATE_ALGORITHM @RT(15)pPressureLintab @STRUCTURED_TEXT
@RT(0) @RT(47)sv_PressureLintab,sv_rValueMinVoltagePresDetect @RT(9)PU_Task_7 @F @F
@END_Algo

@BEG_Dcl
@RT(16)DclTreeContainer
0
@END_Dcl

@END_Export

@BEG_Export

@BEG_Algo
@POSTUPDATE_ALGORITHM @RT(13)pDitherParams @STRUCTURED_TEXT
@RT(0) @RT(60)sv_bInitStart,sv_rDitherAmplitudePres,sv_rDitherAmplitudeVel @RT(9)PU_Task_7 @F @F
@END_Algo

@BEG_Dcl
@RT(16)DclTreeContainer
5
@Var @RT(10)HandleData @RT(0) @T @T @DERIVED 0 @T @T @DT @RT(15)KCAT_HandleData @RT(0) @T @T @UNKNOWN 0 @F
@F @F
@T
@BEG_Attrib
3 @RT(0) @RT(0) @RT(0)
@END_Attrib
1 0 @F @F @F @F

@Var @RT(9)CatStatus @RT(0) @T @T @DERIVED 0 @T @T @DT @RT(11)KCAT_Status @RT(0) @T @T @UNKNOWN 0 @F
@F @F
@T
@BEG_Attrib
3 @RT(0) @RT(0) @RT(0)
@END_Attrib
1 0 @F @F @F @F

@Var @RT(7)sDevice @RT(0) @T @F @DT @RT(10)STRING(31) @RT(0) @T @T @STRING 0 @F @RT(2)31 @F
@F @F
@T
@BEG_Attrib
3 @RT(0) @RT(0) @RT(0)
@END_Attrib
1 0 @F @F @F @F

@Var @RT(9)bInitDone @RT(0) @T @F @DT @RT(4)BOOL @RT(0) @T @T @BASIC 0 @F
@F @F
@T
@BEG_Attrib
3 @RT(0) @RT(0) @RT(0)
@END_Attrib
1 0 @F @F @F @F

@Var @RT(14)bCurrentOutput @RT(0) @T @F @DT @RT(4)BOOL @RT(0) @T @T @BASIC 0 @F
@F @F
@T
@BEG_Attrib
3 @RT(0) @RT(30)TRUE: current output available @RT(0)
@END_Attrib
1 0 @F @F @F @F

@END_Dcl

@END_Export

@BEG_Export

@BEG_Algo
@POSTUPDATE_ALGORITHM @RT(14)pSetMinVoltage @STRUCTURED_TEXT
@RT(0) @RT(79)sv_bInitDone,sv_rMinVoltageVelOutput,sv_rMinVoltagePressOutput,sv_OperationMode @RT(9)PU_Task_3 @F @F
@END_Algo

@BEG_Dcl
@RT(16)DclTreeContainer
0
@END_Dcl

@END_Export

@BEG_Body
@TL(25)
(**************************************** WARNING ********************************************
 *** The KEBA Kemro K2 System including software is not intended for safety control tasks! ***
 ***                       For further information see Comment tab!                        ***
 *********************************************************************************************)

mbStop := FALSE;
//make sure when we get a start and a stop very fast,
//we do not end up in a situation where mbStopped is FALSE but paXxxOutput is still running
mbStopped := FALSE;

abAnalogOutputP.aInit(pLintab := pLintabP);
abAnalogOutputV.aInit(pLintab := pLintabV);

mprPressureSource := prPressure;
mprVelocitySource := prVelocity;

CASE AnaOutMode OF

   nAnaOutputModeMid:
         START_PROCESS_ALGORITHM(paMidOutput);

   nAnaOutputModeFast:
         START_PROCESS_ALGORITHM(paFastOutput);
END_CASE;

@END_Body

@@@BEG_Comment@@@
@TL(0)

@@@END_Comment@@@

@BEG_Body
@TL(10)
(**************************************** WARNING ********************************************
 *** The KEBA Kemro K2 System including software is not intended for safety control tasks! ***
 ***                       For further information see Comment tab!                        ***
 *********************************************************************************************)

IF NOT mbStopped THEN
   mbStop := TRUE;
END_IF;
bReady := mbStopped;

@END_Body

@@@BEG_Comment@@@
@TL(0)

@@@END_Comment@@@

@BEG_Body
@TL(28)
(**************************************** WARNING ********************************************
 *** The KEBA Kemro K2 System including software is not intended for safety control tasks! ***
 ***                       For further information see Comment tab!                        ***
 *********************************************************************************************)

IF NOT abAnalogHWOutV.aIsLinked() THEN
   SET_ALARM(Name := erVariableNotLinked,
             SubID1 := sv_DeviceId.CompId,
             SubID2 := sv_DeviceId.IndexId,
             Param1 := 'ao_Velocity');
END_IF;

IF NOT abAnalogHWOutP.aIsLinked() THEN
   SET_ALARM(Name := erVariableNotLinked,
             SubID1 := sv_DeviceId.CompId,
             SubID2 := sv_DeviceId.IndexId,
             Param1 := 'ao_Pressure');
END_IF;

IF abAnalogOutputP.aRun.bError THEN
   fbDebugTrace(CONCAT('ABPumpOutput: error ',DINT_TO_STRING(abAnalogOutputP.aRun.iErrorInfo),' in ABAnalogOutputP'));
END_IF;

IF abAnalogOutputV.aRun.bError THEN
   fbDebugTrace(CONCAT('ABPumpOutput: error ',DINT_TO_STRING(abAnalogOutputV.aRun.iErrorInfo),' in ABAnalogOutputV'));
END_IF;

@END_Body

@@@BEG_Comment@@@
@TL(0)

@@@END_Comment@@@

@BEG_SfcBody
10 7 8

@BEG_SfcData 2
@StepSeq @RT(4)sseq @F 5
@Step @RT(3)OUT @F @T @T @F @RT(0) @F
@AcbCont @RT(7)unnamed @F 3
@Acb @RT(4)Init @F @T @RT(1)P @RT(0) @F @F @T @TL(2)
mbStopped := FALSE;

@F
@Acb @RT(13)ADitherSignal @F @F @RT(1)N @RT(0) @F @F @F @F
@Acb @RT(4)AOUT @F @T @RT(1)N @RT(0) @F @F @T @TL(14)
//limit pressure output to max. pressure of the pump
rPressure := MIN(sv_rMaxPressure, mprPressureSource^);

b := WRITE_SVREAL_DIRECT(sv_rPressure, rPressure);
b := WRITE_SVREAL_DIRECT(sv_rVelocity, mprVelocitySource^);

(* Lintab Calculation *)
abAnalogOutputP.aRun(rSetValue := sv_rPressure);
abAnalogOutputV.aRun(rSetValue := sv_rVelocity);

(* Output to AO and Shortcircuit detection *)
abAnalogHWOutP.aOut(rValue := (MAX(abAnalogOutputP.aRun.rOutput, mrMinVoltagePressureOutput)) + rDitherPres);
abAnalogHWOutV.aOut(rValue := (MAX(abAnalogOutputV.aRun.rOutput, mrMinVoltageVelocityOutput)) + rDitherVel);

@F

@AltBranch @RT(3)alt @F 2
@TransSeq @RT(4)tseq @F 3
@Trans @RT(6)Trans1 @F @T @F @F @T @T @TL(5)
abAnalogOutputP.aRun.bError OR
abAnalogOutputV.aRun.bError OR
abAnalogHWOutP.aOut.bError OR
abAnalogHWOutV.aOut.bError

@RT(6)Trans1 @F
@Step @RT(10)ERROR_STOP @F @F @F @F @RT(0) @F
@AcbCont @RT(7)unnamed @F 1
@Acb @RT(10)AErrorStop @F @T @RT(1)P @RT(0) @F @F @T @TL(4)
sv_rPressure := 0.0;
sv_rVelocity := 0.0;
aSetErrorMessage();

@F

@Trans @RT(6)Trans5 @F @T @F @F @T @F @TL(2)
TRUE

@RT(6)Trans5 @F

@TransSeq @RT(4)tseq @F 1
@Trans @RT(5)TStop @F @T @T @F @T @F @TL(2)
mbStop

@RT(6)Trans4 @F

@Step @RT(6)S_Stop @F @F @F @F @RT(0) @F
@AcbCont @RT(7)unnamed @F 1
@Acb @RT(5)AStop @F @T @RT(1)P @RT(0) @F @F @T @TL(9)
mbStop := FALSE;

(* Stopping Analog Output*)
abAnalogHWOutP.aOut(rValue := mrMinVoltagePressureOutput);
abAnalogHWOutV.aOut(rValue := mrMinVoltageVelocityOutput);

mbStopped := TRUE;
STOP_PROCESS_ALGORITHM();

@F

@Trans @RT(10)TNewOutput @F @T @F @F @T @T @TL(2)
TRUE

@RT(6)Trans7 @F
@Goto @RT(3)OUT @F @F
@END_SfcData
@SaActions 1
@SaText @RT(13)ADitherSignal 1 @TL(22)
(**************************************** WARNING ********************************************
 *** The KEBA Kemro K2 System including software is not intended for safety control tasks! ***
 ***                       For further information see Comment tab!                        ***
 *********************************************************************************************)

//sinus signals for pressure and velocity dither
IF sv_rDitherAmplitudeVel > 0.0 THEN
   fbSinusVel(rAmplitude := sv_rDitherAmplitudeVel,
              rFrequency := sv_rDitherFrequencyVel,
              rOut => rDitherVel);
ELSE
   rDitherVel := 0.0;
END_IF;

IF sv_rDitherAmplitudePres > 0.0 THEN
   fbSinusPres(rAmplitude := sv_rDitherAmplitudePres,
              rFrequency := sv_rDitherFrequencyPres,
              rOut => rDitherPres);
ELSE
   rDitherPres := 0.0;
END_IF;

@SaTrans 0
@SaExits 0
@END_SfcBody

@@@BEG_Comment@@@
@TL(0)

@@@END_Comment@@@

@BEG_SfcBody
11 8 8

@BEG_SfcData 2
@StepSeq @RT(4)sseq @F 5
@Step @RT(3)OUT @F @T @T @F @RT(0) @F
@AcbCont @RT(7)unnamed @F 3
@Acb @RT(4)Init @F @T @RT(1)P @RT(0) @F @F @T @TL(2)
mbStopped := FALSE;

@F
@Acb @RT(13)ADitherSignal @F @F @RT(1)N @RT(0) @F @F @F @F
@Acb @RT(4)AOUT @F @T @RT(1)N @RT(0) @F @F @T @TL(16)
//limit pressure output to max. pressure of the pump
rPressure := MIN(sv_rMaxPressure, mprPressureSource^);

b := WRITE_SVREAL_DIRECT(sv_rPressure, rPressure);
b := WRITE_SVREAL_DIRECT(sv_rVelocity, mprVelocitySource^);

(* Lintab Calculation *)
abAnalogOutputP.aRun(rSetValue := sv_rPressure);
abAnalogOutputV.aRun(rSetValue := sv_rVelocity);

(* Shortcircuit detection *)
abAnalogHWOutP.aOut(rValue := (MAX(abAnalogOutputP.aRun.rOutput, mrMinVoltagePressureOutput)) + rDitherPres);
abAnalogHWOutV.aOut(rValue := (MAX(abAnalogOutputV.aRun.rOutput, mrMinVoltageVelocityOutput)) + rDitherVel);

@F

@AltBranch @RT(3)alt @F 2
@TransSeq @RT(4)tseq @F 3
@Trans @RT(6)Trans1 @F @T @F @F @T @T @TL(5)
abAnalogOutputP.aRun.bError OR
abAnalogOutputV.aRun.bError OR
abAnalogHWOutP.aOut.bError OR
abAnalogHWOutV.aOut.bError

@RT(6)Trans1 @F
@Step @RT(10)ERROR_STOP @F @F @F @F @RT(0) @F
@AcbCont @RT(7)unnamed @F 1
@Acb @RT(10)AErrorStop @F @T @RT(1)P @RT(0) @F @F @T @TL(4)
sv_rPressure := 0.0;
sv_rVelocity := 0.0;
aSetErrorMessage();

@F

@Trans @RT(6)Trans5 @F @T @F @F @T @F @TL(2)
TRUE

@RT(6)Trans5 @F

@TransSeq @RT(4)tseq @F 1
@Trans @RT(5)TStop @F @T @T @F @T @F @TL(2)
mbStop

@RT(6)Trans4 @F

@Step @RT(6)S_Stop @F @F @F @F @RT(0) @F
@AcbCont @RT(7)unnamed @F 1
@Acb @RT(5)AStop @F @T @RT(1)P @RT(0) @F @F @T @TL(9)
mbStop := FALSE;

(* Stopping Analog Output*)
abAnalogHWOutP.aOut(rValue := mrMinVoltagePressureOutput);
abAnalogHWOutV.aOut(rValue := mrMinVoltageVelocityOutput);

mbStopped := TRUE;
STOP_PROCESS_ALGORITHM();

@F

@Trans @RT(10)TNewOutput @F @T @F @F @T @T @TL(2)
TRUE

@RT(6)Trans7 @F
@Goto @RT(3)OUT @F @F
@END_SfcData
@SaActions 1
@SaText @RT(13)ADitherSignal 1 @TL(22)
(**************************************** WARNING ********************************************
 *** The KEBA Kemro K2 System including software is not intended for safety control tasks! ***
 ***                       For further information see Comment tab!                        ***
 *********************************************************************************************)

//sinus signals for pressure and velocity dither
IF sv_rDitherAmplitudeVel > 0.0 THEN
   fbSinusVel(rAmplitude := sv_rDitherAmplitudeVel,
              rFrequency := sv_rDitherFrequencyVel,
              rOut => rDitherVel);
ELSE
   rDitherVel := 0.0;
END_IF;

IF sv_rDitherAmplitudePres > 0.0 THEN
   fbSinusPres(rAmplitude := sv_rDitherAmplitudePres,
              rFrequency := sv_rDitherFrequencyPres,
              rOut => rDitherPres);
ELSE
   rDitherPres := 0.0;
END_IF;

@SaTrans 0
@SaExits 0
@END_SfcBody

@@@BEG_Comment@@@
@TL(0)

@@@END_Comment@@@

@BEG_Body
@TL(28)
fuName := GET_MY_FU_NAME();
variableName := CONCAT(fuName,'.rPressure Hydr bar');
swoState := KSWO_AddVariable( Task := TaskInject,
                              Name := variableName,
                              Variable := sv_rPressure);
b := FAddToScopeGroup(Task := TaskInject,
                      Name := variableName,
                      GroupId := cScopeGroupPump);
variableName := CONCAT(fuName,'.rVelocity %');
swoState := KSWO_AddVariable( Task := TaskInject,
                              Name := variableName,
                              Variable := sv_rVelocity);
b := FAddToScopeGroup(Task := TaskInject,
                      Name := variableName,
                      GroupId := cScopeGroupPump);

variableName := CONCAT(fuName,'.rPressure Hydr bar');
swoState := KSWO_AddVariable( Task := TaskAnalog,
                              Name := variableName,
                              Variable := sv_rPressure);
variableName := CONCAT(fuName,'.rVelocity %');
swoState := KSWO_AddVariable( Task := TaskAnalog,
                              Name := variableName,
                              Variable := sv_rVelocity);

STOP_PROCESS_ALGORITHM();

@END_Body

@@@BEG_Comment@@@
@TL(0)

@@@END_Comment@@@

@BEG_Body
@TL(26)
(**************************************** WARNING ********************************************
 *** The KEBA Kemro K2 System including software is not intended for safety control tasks! ***
 ***                       For further information see Comment tab!                        ***
 *********************************************************************************************)

LintabParams.LintabPoints := pLintab^.LintabPoints;
LintabParams.Mode.bLinearExtrapolation := TRUE;
LintabParams.Mode.bSetNegativeValuesToZero := FALSE;
LintabParams.Mode.bZeroExtrapolation := FALSE;
Lintab.Par(Param := LintabParams);

IF Lintab.Par.parStatus <> KCTRL_Ret_OK THEN
   rMinVoltage := 0.0;
   RETURN; //error -> return 0.0
END_IF;

//calculate value
Lintab.Calculate(rX := rXValue);
IF Lintab.Calculate.calcStatus <> KCTRL_Ret_OK THEN
   rMinVoltage := 0.0;
   RETURN; //error -> return 0.0
ELSE
   rMinVoltage := Lintab.Calculate.rY;
END_IF;

@END_Body

@@@BEG_Comment@@@
@TL(0)

@@@END_Comment@@@

@BEG_Body
@TL(9)
(**************************************** WARNING ********************************************
 *** The KEBA Kemro K2 System including software is not intended for safety control tasks! ***
 ***                       For further information see Comment tab!                        ***
 *********************************************************************************************)

aGetMinVoltage(pLintab := @sv_VelocityLintab,
               rXValue := sv_rValueMinVoltageVelDetect,
               rMinVoltage => sv_rMinVoltageVelOutput);

@END_Body

@@@BEG_Comment@@@
@TL(0)

@@@END_Comment@@@

@BEG_Body
@TL(9)
(**************************************** WARNING ********************************************
 *** The KEBA Kemro K2 System including software is not intended for safety control tasks! ***
 ***                       For further information see Comment tab!                        ***
 *********************************************************************************************)

aGetMinVoltage(pLintab := @sv_PressureLintab,
               rXValue := sv_rValueMinVoltagePresDetect,
               rMinVoltage => sv_rMinVoltagePressOutput);

@END_Body

@@@BEG_Comment@@@
@TL(0)

@@@END_Comment@@@

@BEG_Body
@TL(29)
(**************************************** WARNING ********************************************
 *** The KEBA Kemro K2 System including software is not intended for safety control tasks! ***
 ***                       For further information see Comment tab!                        ***
 *********************************************************************************************)

IF NOT bInitDone THEN
   //get device name
   HandleData := KCAT_GetHandle('IO.ONBOARD.deviceName');
   IF HandleData.Status = KCAT_Status_OK THEN
      CatStatus := KCAT_GetValue(Handle := HandleData.Handle, Buffer := sDevice);
      sDevice := LEFT(sDevice,5);

      IF sDevice ='CP 03' THEN
         bCurrentOutput := TRUE;
      END_IF;
   END_IF;

   bInitDone := TRUE;

END_IF;

IF NOT bCurrentOutput THEN
   //set dither amplitude to 0.0 (=disable dither signal)
   sv_rDitherAmplitudeVel := 0.0;
   sv_rDitherAmplitudePres := 0.0;
END_IF;

@END_Body

@@@BEG_Comment@@@
@TL(0)

@@@END_Comment@@@

@BEG_Body
@TL(22)
(**************************************** WARNING ********************************************
 *** The KEBA Kemro K2 System including software is not intended for safety control tasks! ***
 ***                       For further information see Comment tab!                        ***
 *********************************************************************************************)

IF sv_OperationMode = nSetup THEN
   //setup mode -> set minimum output voltage to 0.0
   mrMinVoltagePressureOutput := 0.0;
   mrMinVoltageVelocityOutput := 0.0;

ELSE
   //all other operation modes
   mrMinVoltagePressureOutput := sv_rMinVoltagePressOutput;
   mrMinVoltageVelocityOutput := sv_rMinVoltageVelOutput;
END_IF;

IF mbStopped THEN
   //write to AO´s immediately if device is not active
   abAnalogHWOutP.aOut(rValue := mrMinVoltagePressureOutput);
   abAnalogHWOutV.aOut(rValue := mrMinVoltageVelocityOutput);
END_IF;

@END_Body

@@@BEG_Comment@@@
@TL(0)

@@@END_Comment@@@
@END_Body

@END_Contents

(* ---- ABPumpPressureCalibCycle.pu ---- *)
(*
Do steps for automatic Pump pressure calibration
*)

IMPORT_OVER_LISTFILE
 SET_ALARM
, SET_EVENT
, START_PROCESS_ALGORITHM
, tnCalibState_Running
, cCalibFilePres
, tnOperationMode
, tsCalibMovement
, KAPPL_LintabData3D
, tyPumpData
, tevStartRequest
, ABAutoCalibRedoListener
, FBCalibWriteLog
, tsTraceLevel
, KAPPL_LintabData
, tsPumpCalibError
, tsDeviceId
, tMoveIdent
, tsRequiredPumps
, tyCalibDevices
, tevStartRequestData
, FBCheckReady
, FBStopStartedMovements
, FBAutoCalibLog
, TON
, tyRequiredPumps
, ABCreateMeasureArray

END_IMPORT

ALGORITHM_BLOCK ABPumpPressureCalibCycle #DUMMY_EDIT_BLOCK

SYSTEM_VAR
 sv_OperationMode : tnOperationMode;
 sv_bPumpPreVelCalibDone : BOOL;
 sv_bPumpPreVelCalibAnotherStepN : BOOL;
 sv_CalibStatePumpPressure : tsCalibMovement;
 sv_bDoPumpPressureCalib : BOOL;
 sv_TmpLintab : KAPPL_LintabData3D;
 sv_PumpData : tyPumpData;
 sv_TraceLevel : tsTraceLevel;
 sv_dDelayTimeNextShot : TIME;
 sv_PressureLintab : KAPPL_LintabData;
 sv_PumpCalibError : tsPumpCalibError;
 sv_iCalibratingPump : DINT (* number of pump which is actually calibrating *);
 sv_DeviceId : tsDeviceId;
 sv_bInitDone : BOOL;
 sv_iDeviceForCalib : DINT;
 sv_PumpCalibDevices : tyCalibDevices (* !!! device 1 - 20 reserved !!! *);
END_VAR

SYSTEM_OBJECT
 TaskMid : TASK;
 PU_Task_7 : TASK;
 evStartRequest : tevStartRequest;
 erHighDiffAtPres : ALARM;
 TaskSlow : TASK;
 erPumpPresCalibNoValueChange : ALARM;
 erCalibrationPressureNotStable : ALARM;
 PU_Task_13 : TASK;
END_OBJECT

VAR
 abAutoCalibRedoListenerPressure : ABAutoCalibRedoListener;
 fbCalibWriteLog : FBCalibWriteLog;
 mbFilesDeleted : BOOL;
 mbLogFileSaved : BOOL := TRUE;
 mpbCalibError : REFTO BOOL;
 mMoveIdStartPos : tMoveIdent (* move id of the movement which must be started to move to pressure calib start position *);
 mMoveDirStartPos : tMoveIdent (* move direction of the movement which must be started to move to pressure calib start position *);
 mMoveDirCalib : tMoveIdent (* move direction of calibration movement *);
 mMoveIdCalib : tMoveIdent (* move id of calibration movement *);
 mpRequiredPumps : REFTO tsRequiredPumps;
 mDeviceForCalib : tsDeviceId;
END_VAR

POSTUPDATE_ALGORITHM pStart ON PU_Task_7 WITH sv_CalibStatePumpPressure.Status

#BEGIN_EDIT_BLOCK
(**************************************** WARNING ********************************************
 *** The KEBA Kemro K2 System including software is not intended for safety control tasks! ***
 ***                       For further information see Comment tab!                        ***
 *********************************************************************************************)

IF sv_OperationMode = nSetup THEN
   IF sv_CalibStatePumpPressure.Status = tnCalibState_Running THEN
      IF sv_CalibStatePumpPressure.Group = tnCalibGroup_LintabOnly THEN
         //do not start pump calibration and set calib state to "done"
         sv_CalibStatePumpPressure.Status := tnCalibState_Done;
      ELSE
         sv_PumpCalibError.bError := FALSE;
         sv_PumpCalibError.iErrorInfo := 0;
         mpbCalibError := @sv_PumpCalibError.bError;
         START_PROCESS_ALGORITHM(paRun);
      END_IF;
   END_IF;
END_IF;

;#END_EDIT_BLOCK END_ALGORITHM

PROCESS_ALGORITHM paRun ON TaskMid

VAR_TEMP
 uTmpCnt : UDINT;
END_VAR

VAR
 evStartRequestData : tevStartRequestData;
 fbCheckReady : FBCheckReady;
 fbStopStartedMovements : FBStopStartedMovements;
 fbLog : FBAutoCalibLog;
 rMaxDetectPressure : REAL (* Maximal identified pressure *);
 rMinFac : REAL := 0.05 (* security factor for checking difference of detected pressure and max. pressure *);
 DelayTimer : TON;
 OriginalPumpAssignment : tyRequiredPumps;
 NoAssignedPumps : tyRequiredPumps;
 tmpAssignment : tyRequiredPumps;
 rMaxPressure : REAL;
 abCreateMeasureArray : ABCreateMeasureArray;
END_VAR

(* IecGraph-Code *)

(* init step *)
INITIAL_STEP S_INIT:
AInit (P);
APumpAssignment (P);
END_STEP

ACTION AInit: #BEGIN_EDIT_BLOCK
sv_bDoPumpPressureCalib := TRUE;
sv_bPumpPreVelCalibAnotherStepN := FALSE;
sv_bPumpPreVelCalibDone := FALSE;
sv_iCalibratingPump := sv_DeviceId.IndexId;
sv_CalibStatePumpPressure.prGlobalMaxX^ := sv_PumpData[sv_DeviceId.IndexId].prMaxPressure^;
sv_CalibStatePumpPressure.prGlobalMaxY^ := 10.0; //V

abCreateMeasureArray.aInit();  //create dynamic arrays
fbLog('pressure calib started');

;#END_EDIT_BLOCK END_ACTION (*AInit*)
ACTION APumpAssignment: #BEGIN_EDIT_BLOCK
//save actual pump assigment
OriginalPumpAssignment := mpRequiredPumps^.RequiredPumps;

//change assignment to the pump which should be calibrated
tmpAssignment := NoAssignedPumps;
tmpAssignment[sv_iCalibratingPump] := TRUE;
mpRequiredPumps^.RequiredPumps := tmpAssignment;

;#END_EDIT_BLOCK END_ACTION (*APumpAssignment*)

(* steps *)
STEP S_RESET:
AStopmovements (P);
Action24 (P);
AWaitReady (N);
END_STEP

ACTION Action24: #BEGIN_EDIT_BLOCK
IF sv_CalibStatePumpPressure.Status <> tnCalibState_Error THEN
   fbLog('pressure calib aborted');
   sv_CalibStatePumpPressure.Status := tnCalibState_Aborted;
ELSE
   fbLog('pressure calib failure');
END_IF;

;#END_EDIT_BLOCK END_ACTION (*Action24*)
ACTION AWaitReady: #BEGIN_EDIT_BLOCK
fbCheckReady(DeviceId := mDeviceForCalib);

;#END_EDIT_BLOCK END_ACTION (*AWaitReady*)
STEP S_STOP:
Action22 (P);
END_STEP

ACTION Action22: #BEGIN_EDIT_BLOCK
sv_bDoPumpPressureCalib := FALSE;
mpbCalibError := EMPTY;
sv_iCalibratingPump := 0;
//restore original assignment
mpRequiredPumps^.RequiredPumps := OriginalPumpAssignment;

//delete dynamic arrays
abCreateMeasureArray.aRelease();

STOP_PROCESS_ALGORITHM();

;#END_EDIT_BLOCK END_ACTION (*Action22*)
STEP Step10:
Delete_LogFiles (P);
END_STEP

STEP S_StartPos:
AMoveStartPos (P);
Action8 (N);
END_STEP

ACTION Action8: #BEGIN_EDIT_BLOCK
fbCheckReady(DeviceId := mDeviceForCalib);

;#END_EDIT_BLOCK END_ACTION (*Action8*)
STEP S_Calib:
ACalib (P);
Action9 (N);
END_STEP

ACTION Action9: #BEGIN_EDIT_BLOCK
fbCheckReady(DeviceId := mDeviceForCalib);

;#END_EDIT_BLOCK END_ACTION (*Action9*)
STEP S_WAIT_CALC:
Action27 (P);
END_STEP

ACTION Action27: #BEGIN_EDIT_BLOCK
//show lintab during calibration
sv_CalibStatePumpPressure.pDisplayLintab^.LintabPoints.uNoOfPoints := sv_TmpLintab.LintabPoints.uNoOfPoints;
FOR uTmpCnt := 1 TO sv_TmpLintab.LintabPoints.uNoOfPoints DO
   sv_CalibStatePumpPressure.pDisplayLintab^.LintabPoints.Point[uTmpCnt].rX:= sv_TmpLintab.LintabPoints.Point[uTmpCnt].rX;
   sv_CalibStatePumpPressure.pDisplayLintab^.LintabPoints.Point[uTmpCnt].rY:= sv_TmpLintab.LintabPoints.Point[uTmpCnt].rY;
END_FOR;
DelayTimer(IN:=FALSE);
DelayTimer(IN:=TRUE, PT:=sv_dDelayTimeNextShot);

;#END_EDIT_BLOCK END_ACTION (*Action27*)
STEP Step11:
Write_LogFile (P);
END_STEP

STEP Step12:
WaitDelay (N);
END_STEP

ACTION WaitDelay: #BEGIN_EDIT_BLOCK
DelayTimer(IN:=TRUE);

;#END_EDIT_BLOCK END_ACTION (*WaitDelay*)
STEP S_DONE:
Action18 (P);
ACompareToMaxPressure (P);
END_STEP

ACTION Action18: #BEGIN_EDIT_BLOCK
//copy lintab and set calib state
fbLog('pressure calib finished');
sv_PressureLintab := sv_CalibStatePumpPressure.pDisplayLintab^;
sv_CalibStatePumpPressure.Status := tnCalibState_Done;

;#END_EDIT_BLOCK END_ACTION (*Action18*)

(* transitions *)
TRANSITION TCalibDeviceReady (* Trans15 *) FROM S_RESET TO S_STOP :=  #BEGIN_EDIT_BLOCK
fbCheckReady.bReady AND mbLogFileSaved
;#END_EDIT_BLOCK
END_TRANSITION

TRANSITION Trans18 (* Trans18 *) FROM S_STOP TO S_INIT :=  #BEGIN_EDIT_BLOCK
TRUE
;#END_EDIT_BLOCK
END_TRANSITION

TRANSITION Trans1 (* Trans1 *) FROM S_INIT TO Step10 :=  #BEGIN_EDIT_BLOCK
sv_TraceLevel.bDebugCalibration

;#END_EDIT_BLOCK
END_TRANSITION

TRANSITION Trans10 (* Trans10 *) FROM Step10 TO S_StartPos :=  #BEGIN_EDIT_BLOCK
mbFilesDeleted
;#END_EDIT_BLOCK
END_TRANSITION

TRANSITION Trans13 (* Trans13 *) FROM S_INIT TO S_StartPos :=  #BEGIN_EDIT_BLOCK
NOT sv_TraceLevel.bDebugCalibration
;#END_EDIT_BLOCK
END_TRANSITION

TRANSITION Trans5 (* Trans5 *) FROM S_StartPos TO S_Calib :=  #BEGIN_EDIT_BLOCK
fbCheckReady.bReady
;#END_EDIT_BLOCK
END_TRANSITION

TRANSITION Trans2 (* Trans2 *) FROM S_Calib TO S_WAIT_CALC :=  #BEGIN_EDIT_BLOCK
fbCheckReady.bReady
;#END_EDIT_BLOCK
END_TRANSITION

TRANSITION Trans14 (* Trans14 *) FROM S_WAIT_CALC TO Step11 :=  #BEGIN_EDIT_BLOCK
sv_TraceLevel.bDebugCalibration
;#END_EDIT_BLOCK
END_TRANSITION

TRANSITION Trans30 (* Trans15 *) FROM Step11 TO Step12 :=  #BEGIN_EDIT_BLOCK
mbLogFileSaved
;#END_EDIT_BLOCK
END_TRANSITION

TRANSITION Trans16 (* Trans16 *) FROM S_WAIT_CALC TO Step12 :=  #BEGIN_EDIT_BLOCK
NOT sv_TraceLevel.bDebugCalibration
;#END_EDIT_BLOCK
END_TRANSITION

TRANSITION Trans24 (* Trans24 *) FROM Step12 TO S_Calib :=  #BEGIN_EDIT_BLOCK
sv_bPumpPreVelCalibAnotherStepN AND
DelayTimer.Q
// another step needed
;#END_EDIT_BLOCK
END_TRANSITION

TRANSITION Trans21 (* Trans21 *) FROM Step12 TO S_DONE :=  #BEGIN_EDIT_BLOCK
sv_bPumpPreVelCalibDone
//calib finished
;#END_EDIT_BLOCK
END_TRANSITION

TRANSITION Trans23 (* Trans23 *) FROM Step12 TO S_RESET :=  #BEGIN_EDIT_BLOCK
NOT sv_bPumpPreVelCalibAnotherStepN
AND NOT sv_bPumpPreVelCalibDone
//maybe remove in vlavour of exit
;#END_EDIT_BLOCK
END_TRANSITION

TRANSITION Trans19 (* Trans19 *) FROM S_DONE TO S_STOP :=  #BEGIN_EDIT_BLOCK
TRUE
;#END_EDIT_BLOCK
END_TRANSITION

(* end IecGraph-Code *)
(* sfc-code *)

(* stand alone actions *)
ACTION AMoveStartPos: #BEGIN_EDIT_BLOCK
(**************************************** WARNING ********************************************
 *** The KEBA Kemro K2 System including software is not intended for safety control tasks! ***
 ***                       For further information see Comment tab!                        ***
 *********************************************************************************************)

evStartRequestData.DeviceId := mDeviceForCalib;
evStartRequestData.MoveDir := mMoveDirStartPos;
evStartRequestData.MoveId := mMoveIdStartPos;
SET_EVENT(evStartRequest, evStartRequestData);

;#END_EDIT_BLOCK END_ACTION (*AMoveStartPos*)
ACTION AStopmovements: #BEGIN_EDIT_BLOCK
(**************************************** WARNING ********************************************
 *** The KEBA Kemro K2 System including software is not intended for safety control tasks! ***
 ***                       For further information see Comment tab!                        ***
 *********************************************************************************************)

fbStopStartedMovements();

;#END_EDIT_BLOCK END_ACTION (*AStopmovements*)
ACTION ACalib: #BEGIN_EDIT_BLOCK
(**************************************** WARNING ********************************************
 *** The KEBA Kemro K2 System including software is not intended for safety control tasks! ***
 ***                       For further information see Comment tab!                        ***
 *********************************************************************************************)

evStartRequestData.DeviceId := mDeviceForCalib;
evStartRequestData.MoveDir := mMoveDirCalib;
evStartRequestData.MoveId := mMoveIdCalib;
SET_EVENT(evStartRequest, evStartRequestData);

;#END_EDIT_BLOCK END_ACTION (*ACalib*)
ACTION ACompareToMaxPressure: #BEGIN_EDIT_BLOCK
(**************************************** WARNING ********************************************
 *** The KEBA Kemro K2 System including software is not intended for safety control tasks! ***
 ***                       For further information see Comment tab!                        ***
 *********************************************************************************************)

// Set alarm if detected pressure differs too strong from max. pressure
rMaxDetectPressure := sv_PressureLintab.LintabPoints.Point[sv_PressureLintab.LintabPoints.uNoOfPoints].rX;
rMaxPressure := sv_PumpData[sv_DeviceId.IndexId].prMaxPressure^;
IF ABS(rMaxPressure - rMaxDetectPressure) > (rMinFac * rMaxPressure) THEN
   SET_ALARM(Name := erHighDiffAtPres,
             SubID1 := sv_DeviceId.CompId,
             SubID2 := sv_DeviceId.IndexId);
END_IF;

;#END_EDIT_BLOCK END_ACTION (*ACompareToMaxPressure*)
ACTION Delete_LogFiles: #BEGIN_EDIT_BLOCK
(**************************************** WARNING ********************************************
 *** The KEBA Kemro K2 System including software is not intended for safety control tasks! ***
 ***                       For further information see Comment tab!                        ***
 *********************************************************************************************)

mbFilesDeleted := FALSE;
START_PROCESS_ALGORITHM(paDeleteLogFiles);

;#END_EDIT_BLOCK END_ACTION (*Delete_LogFiles*)
ACTION Write_LogFile: #BEGIN_EDIT_BLOCK
(**************************************** WARNING ********************************************
 *** The KEBA Kemro K2 System including software is not intended for safety control tasks! ***
 ***                       For further information see Comment tab!                        ***
 *********************************************************************************************)

mbLogFileSaved := FALSE;
START_PROCESS_ALGORITHM(paWriteLogFile);

;#END_EDIT_BLOCK END_ACTION (*Write_LogFile*)

(* exits *)

EXIT_TRANSITION E_NotSetupMode := #BEGIN_EDIT_BLOCK
(**************************************** WARNING ********************************************
 *** The KEBA Kemro K2 System including software is not intended for safety control tasks! ***
 ***                       For further information see Comment tab!                        ***
 *********************************************************************************************)

sv_OperationMode <> nSetup
;#END_EDIT_BLOCK
PRIORITY 1 WITH  INITIAL_STEP S_RESET: END_STEP
END_TRANSITION

EXIT_TRANSITION E_NotCalibratingAnymore := #BEGIN_EDIT_BLOCK
// abort calibration, when not in running state and not finished
sv_CalibStatePumpPressure.Status <> tnCalibState_Running AND (S_INIT.X OR S_StartPos.X OR S_Calib.X OR S_WAIT_CALC.X)
;#END_EDIT_BLOCK
PRIORITY 1 WITH  INITIAL_STEP S_RESET: END_STEP
END_TRANSITION
(* end sfc-code *)

END_ALGORITHM

PROCESS_ALGORITHM paDeleteLogFiles ON TaskSlow

#BEGIN_EDIT_BLOCK
(**************************************** WARNING ********************************************
 *** The KEBA Kemro K2 System including software is not intended for safety control tasks! ***
 ***                       For further information see Comment tab!                        ***
 *********************************************************************************************)

fbCalibWriteLog(fileName:=cCalibFilePres,bDeleteFiles:=TRUE);
mbFilesDeleted := TRUE;
STOP_PROCESS_ALGORITHM();

;#END_EDIT_BLOCK END_ALGORITHM

PROCESS_ALGORITHM paWriteLogFile ON TaskSlow

#BEGIN_EDIT_BLOCK
(**************************************** WARNING ********************************************
 *** The KEBA Kemro K2 System including software is not intended for safety control tasks! ***
 ***                       For further information see Comment tab!                        ***
 *********************************************************************************************)

fbCalibWriteLog(fileName:= cCalibFilePres,bDeleteFiles := FALSE);
mbLogFileSaved := TRUE;
STOP_PROCESS_ALGORITHM();

;#END_EDIT_BLOCK END_ALGORITHM

POSTUPDATE_ALGORITHM pPumpCalibError ON PU_Task_7 WITH mpbCalibError^

#BEGIN_EDIT_BLOCK
(**************************************** WARNING ********************************************
 *** The KEBA Kemro K2 System including software is not intended for safety control tasks! ***
 ***                       For further information see Comment tab!                        ***
 *********************************************************************************************)

IF sv_PumpCalibError.bError THEN

   sv_CalibStatePumpPressure.Status := tnCalibState_Error;
   IF sv_PumpCalibError.iErrorInfo = cValueChangeDuringCalibTooLow THEN
      SET_ALARM(erPumpPresCalibNoValueChange);
   ELSE
      SET_ALARM(erCalibrationPressureNotStable);
   END_IF;

END_IF;

;#END_EDIT_BLOCK END_ALGORITHM

POSTUPDATE_ALGORITHM pInit ON PU_Task_13 WITH sv_bInitDone,sv_iDeviceForCalib

#BEGIN_EDIT_BLOCK
(**************************************** WARNING ********************************************
 *** The KEBA Kemro K2 System including software is not intended for safety control tasks! ***
 ***                       For further information see Comment tab!                        ***
 *********************************************************************************************)

mDeviceForCalib.CompId := cMinCompId;
mDeviceForCalib.IndexId := cMinMoveIdent;
mMoveDirStartPos := cMinMoveIdent;
mMoveIdStartPos := cMinMoveIdent;
mMoveDirCalib := cMinMoveIdent;
mMoveIdCalib := cMinMoveIdent;
mpRequiredPumps := EMPTY;
sv_CalibStatePumpPressure.prInputSensor := EMPTY;
sv_CalibStatePumpPressure.Group := tnCalibGroup_LintabOnly;

IF (sv_iDeviceForCalib > 0) AND (sv_iDeviceForCalib <= cMaxCalibDevices) THEN
   mDeviceForCalib := sv_PumpCalibDevices[sv_iDeviceForCalib].DeviceId;

   IF CHECK_REF(sv_PumpCalibDevices[sv_iDeviceForCalib].pPresCalibStartPosMovement^) THEN
      mMoveDirStartPos := sv_PumpCalibDevices[sv_iDeviceForCalib].pPresCalibStartPosMovement^.MoveDir;
      mMoveIdStartPos :=  sv_PumpCalibDevices[sv_iDeviceForCalib].pPresCalibStartPosMovement^.MoveId;
   END_IF;

   IF CHECK_REF(sv_PumpCalibDevices[sv_iDeviceForCalib].pPresCalibMovement^) THEN
      mMoveDirCalib := sv_PumpCalibDevices[sv_iDeviceForCalib].pPresCalibMovement^.MoveDir;
      mMoveIdCalib := sv_PumpCalibDevices[sv_iDeviceForCalib].pPresCalibMovement^.MoveId;
      mpRequiredPumps := sv_PumpCalibDevices[sv_iDeviceForCalib].pPresCalibMovement^.AnaOutData.pRequiredPumps;
   END_IF;

   IF CHECK_REF(sv_PumpCalibDevices[sv_iDeviceForCalib].prActPressure^) THEN
      sv_CalibStatePumpPressure.prInputSensor := sv_PumpCalibDevices[sv_iDeviceForCalib].prActPressure;
      sv_CalibStatePumpPressure.Group := tnCalibGroup_Pressure;
   END_IF;
END_IF;

;#END_EDIT_BLOCK END_ALGORITHM

END_ALGORITHM_BLOCK

#END_OF_IEC_PART

@Puma @IecEditor 6 103 @Pou 25
@@@BEG_Comment@@@
Do steps for automatic Pump pressure calibration
@@@END_Comment@@@

@BEG_Contents

@BEG_Func
@RT(17)FuncTreeContainer
3
@Var @RT(9)SET_ALARM @RT(0) @T @T @DERIVED 0 @F @RT(23)KEBA_STANDARD_PROCEDURE @F
@T
@BEG_Attrib
0 @RT(0) @RT(0)
@END_Attrib
1 1 @F @F @F @F

@Var @RT(9)SET_EVENT @RT(0) @T @T @DERIVED 0 @F @RT(23)KEBA_STANDARD_PROCEDURE @F
@T
@BEG_Attrib
0 @RT(0) @RT(0)
@END_Attrib
1 1 @F @F @F @F

@Var @RT(23)START_PROCESS_ALGORITHM @RT(0) @T @T @DERIVED 0 @F @RT(23)KEBA_STANDARD_PROCEDURE @F
@T
@BEG_Attrib
0 @RT(0) @RT(0)
@END_Attrib
1 1 @F @F @F @F

@END_Func

@BEG_Const
@RT(18)ConstTreeContainer
2
@Var @RT(20)tnCalibState_Running @RT(0) @T @T @DERIVED 0 @F @RT(12)tnCalibState @F
@T
@BEG_Attrib
0 @RT(1)1 @RT(23)calibration in progress
@END_Attrib
1 1 @F @F @F @F

@Var @RT(14)cCalibFilePres @RT(0) @T @F @DT @RT(11)STRING(255) @RT(0) @T @T @STRING 0 @F @RT(3)255 @F
@F @F
@T
@BEG_Attrib
0 @RT(15)'CalibPumpPres' @RT(42)Filename for Pump Pressure Calib Debug-Log
@END_Attrib
1 1 @F @F @F @F

@END_Const

@BEG_Export

@BEG_Kind
@ALGORITHM_BLOCK @RT(24)ABPumpPressureCalibCycle @STRUCTURED_TEXT
@RT(0) @RT(0) @RT(0)
@END_Kind

@BEG_Dcl
@RT(16)DclTreeContainer
35
@Var @RT(16)sv_OperationMode @RT(0) @T @T @DERIVED 0 @T @T @DT @RT(15)tnOperationMode @RT(0) @T @T @UNKNOWN 0 @F
@F @F
@T
@BEG_Attrib
3 @RT(0) @RT(0) @RT(0)
@END_Attrib
1 8 @F @F @F @F

@Var @RT(23)sv_bPumpPreVelCalibDone @RT(0) @T @F @DT @RT(4)BOOL @RT(0) @T @T @BASIC 0 @F
@F @F
@T
@BEG_Attrib
3 @RT(0) @RT(0) @RT(0)
@END_Attrib
1 8 @F @F @F @F

@Var @RT(31)sv_bPumpPreVelCalibAnotherStepN @RT(0) @T @F @DT @RT(4)BOOL @RT(0) @T @T @BASIC 0 @F
@F @F
@T
@BEG_Attrib
3 @RT(0) @RT(0) @RT(0)
@END_Attrib
1 8 @F @F @F @F

@Var @RT(25)sv_CalibStatePumpPressure @RT(0) @T @T @DERIVED 0 @T @T @DT @RT(15)tsCalibMovement @RT(0) @T @T @UNKNOWN 0 @F
@F @F
@T
@BEG_Attrib
3 @RT(0) @RT(0) @RT(0)
@END_Attrib
1 8 @F @F @F @F

@Var @RT(23)sv_bDoPumpPressureCalib @RT(0) @T @F @DT @RT(4)BOOL @RT(0) @T @T @BASIC 0 @F
@F @F
@T
@BEG_Attrib
3 @RT(0) @RT(0) @RT(0)
@END_Attrib
1 8 @F @F @F @F

@Var @RT(12)sv_TmpLintab @RT(0) @T @T @DERIVED 0 @T @T @DT @RT(18)KAPPL_LintabData3D @RT(0) @T @T @UNKNOWN 0 @F
@F @F
@T
@BEG_Attrib
3 @RT(0) @RT(0) @RT(0)
@END_Attrib
1 8 @F @F @F @F

@Var @RT(11)sv_PumpData @RT(0) @T @T @DERIVED 0 @T @T @DT @RT(10)tyPumpData @RT(0) @T @T @UNKNOWN 0 @F
@F @F
@T
@BEG_Attrib
3 @RT(0) @RT(0) @RT(0)
@END_Attrib
1 8 @F @F @F @F

@Var @RT(7)TaskMid @RT(0) @T @F @DT @RT(4)TASK @RT(0) @T @T @BASIC 0 @F
@F @F
@T
@BEG_Attrib
3 @RT(0) @RT(0) @RT(0)
@END_Attrib
1 7 @F @F @F @F

@Var @RT(9)PU_Task_7 @RT(0) @T @F @DT @RT(4)TASK @RT(0) @T @T @BASIC 0 @F
@F @F
@T
@BEG_Attrib
3 @RT(0) @RT(0) @RT(0)
@END_Attrib
1 7 @F @F @F @F

@Var @RT(14)evStartRequest @RT(0) @T @T @DERIVED 0 @T @T @DT @RT(15)tevStartRequest @RT(0) @T @T @UNKNOWN 0 @F
@F @F
@T
@BEG_Attrib
3 @RT(0) @RT(0) @RT(0)
@END_Attrib
1 7 @F @F @F @F

@Var @RT(16)erHighDiffAtPres @RT(0) @T @F @DT @RT(5)ALARM @RT(0) @T @T @BASIC 0 @F
@F @F
@T
@BEG_Attrib
3 @RT(0) @RT(0) @RT(0)
@END_Attrib
1 7 @F @F @F @F

@Var @RT(31)abAutoCalibRedoListenerPressure @RT(0) @T @T @DERIVED 0 @T @T @DT @RT(23)ABAutoCalibRedoListener @RT(0) @T @T @UNKNOWN 0 @F
@F @F
@T
@BEG_Attrib
3 @RT(0) @RT(0) @RT(0)
@END_Attrib
1 0 @F @F @F @F

@Var @RT(15)fbCalibWriteLog @RT(0) @T @T @DERIVED 0 @T @T @DT @RT(15)FBCalibWriteLog @RT(0) @T @T @UNKNOWN 0 @F
@F @F
@T
@BEG_Attrib
3 @RT(0) @RT(0) @RT(0)
@END_Attrib
1 0 @F @F @F @F

@Var @RT(13)sv_TraceLevel @RT(0) @T @T @DERIVED 0 @T @T @DT @RT(12)tsTraceLevel @RT(0) @T @T @UNKNOWN 0 @F
@F @F
@T
@BEG_Attrib
3 @RT(0) @RT(0) @RT(0)
@END_Attrib
1 8 @F @F @F @F

@Var @RT(8)TaskSlow @RT(0) @T @T @RENAMED 0 @T @T @DT @RT(4)TASK @RT(0) @T @T @BASIC 0 @F
@F @F
@T
@BEG_Attrib
3 @RT(0) @RT(0) @RT(0)
@END_Attrib
1 7 @F @F @F @F

@Var @RT(14)mbFilesDeleted @RT(0) @T @F @DT @RT(4)BOOL @RT(0) @T @T @BASIC 0 @F
@F @F
@T
@BEG_Attrib
3 @RT(0) @RT(0) @RT(0)
@END_Attrib
1 0 @F @F @F @F

@Var @RT(14)mbLogFileSaved @RT(0) @T @F @DT @RT(4)BOOL @RT(0) @T @T @BASIC 0 @F
@F @F
@T
@BEG_Attrib
3 @RT(4)TRUE @RT(0) @RT(0)
@END_Attrib
1 0 @F @F @F @F

@Var @RT(21)sv_dDelayTimeNextShot @RT(0) @T @F @DT @RT(4)TIME @RT(0) @T @T @BASIC 0 @F
@F @F
@T
@BEG_Attrib
3 @RT(0) @RT(0) @RT(0)
@END_Attrib
1 8 @F @F @F @F

@Var @RT(17)sv_PressureLintab @RT(0) @T @T @DERIVED 0 @T @T @DT @RT(16)KAPPL_LintabData @RT(0) @T @T @UNKNOWN 0 @F
@F @F
@T
@BEG_Attrib
3 @RT(0) @RT(0) @RT(0)
@END_Attrib
1 8 @F @F @F @F

@Var @RT(17)sv_PumpCalibError @RT(0) @T @T @DERIVED 0 @T @T @DT @RT(16)tsPumpCalibError @RT(0) @T @T @UNKNOWN 0 @F
@F @F
@T
@BEG_Attrib
3 @RT(0) @RT(0) @RT(0)
@END_Attrib
1 8 @F @F @F @F

@Var @RT(13)mpbCalibError @RT(0) @T @T @REFTO 0 @T @DT @RT(4)BOOL @RT(0) @T @T @BASIC 0 @F
@F @F
@T
@BEG_Attrib
3 @RT(0) @RT(0) @RT(0)
@END_Attrib
1 0 @F @F @F @F

@Var @RT(28)erPumpPresCalibNoValueChange @RT(0) @T @F @DT @RT(5)ALARM @RT(0) @T @T @BASIC 0 @F
@F @F
@T
@BEG_Attrib
3 @RT(0) @RT(0) @RT(0)
@END_Attrib
1 7 @F @F @F @F

@Var @RT(30)erCalibrationPressureNotStable @RT(0) @T @F @DT @RT(5)ALARM @RT(0) @T @T @BASIC 0 @F
@F @F
@T
@BEG_Attrib
3 @RT(0) @RT(0) @RT(0)
@END_Attrib
1 7 @F @F @F @F

@Var @RT(19)sv_iCalibratingPump @RT(0) @T @F @DT @RT(4)DINT @RT(0) @T @T @BASIC 0 @F
@F @F
@T
@BEG_Attrib
3 @RT(0) @RT(44)number of pump which is actually calibrating @RT(0)
@END_Attrib
1 8 @F @F @F @F

@Var @RT(11)sv_DeviceId @RT(0) @T @T @DERIVED 0 @T @T @DT @RT(10)tsDeviceId @RT(0) @T @T @UNKNOWN 0 @F
@F @F
@T
@BEG_Attrib
3 @RT(0) @RT(0) @RT(0)
@END_Attrib
1 8 @F @F @F @F

@Var @RT(12)sv_bInitDone @RT(0) @T @T @RENAMED 0 @T @T @DT @RT(4)BOOL @RT(0) @T @T @BASIC 0 @F
@F @F
@T
@BEG_Attrib
3 @RT(0) @RT(0) @RT(0)
@END_Attrib
1 8 @F @F @F @F

@Var @RT(10)PU_Task_13 @RT(0) @T @T @RENAMED 0 @T @T @DT @RT(4)TASK @RT(0) @T @T @BASIC 0 @F
@F @F
@T
@BEG_Attrib
3 @RT(0) @RT(0) @RT(0)
@END_Attrib
1 7 @F @F @F @F

@Var @RT(15)mMoveIdStartPos @RT(0) @T @T @DERIVED 0 @T @T @DT @RT(10)tMoveIdent @RT(0) @T @T @UNKNOWN 0 @F
@F @F
@T
@BEG_Attrib
3 @RT(0) @RT(86)move id of the movement which must be started to move to pressure calib start position @RT(0)
@END_Attrib
1 0 @F @F @F @F

@Var @RT(16)mMoveDirStartPos @RT(0) @T @T @DERIVED 0 @T @T @DT @RT(10)tMoveIdent @RT(0) @T @T @UNKNOWN 0 @F
@F @F
@T
@BEG_Attrib
3 @RT(0) @RT(93)move direction of the movement which must be started to move to pressure calib start position @RT(0)
@END_Attrib
1 0 @F @F @F @F

@Var @RT(13)mMoveDirCalib @RT(0) @T @T @DERIVED 0 @T @T @DT @RT(10)tMoveIdent @RT(0) @T @T @UNKNOWN 0 @F
@F @F
@T
@BEG_Attrib
3 @RT(0) @RT(38)move direction of calibration movement @RT(0)
@END_Attrib
1 0 @F @F @F @F

@Var @RT(12)mMoveIdCalib @RT(0) @T @T @DERIVED 0 @T @T @DT @RT(10)tMoveIdent @RT(0) @T @T @UNKNOWN 0 @F
@F @F
@T
@BEG_Attrib
3 @RT(0) @RT(31)move id of calibration movement @RT(0)
@END_Attrib
1 0 @F @F @F @F

@Var @RT(15)mpRequiredPumps @RT(0) @T @T @REFTO 0 @F @DERIVED 0 @T @T @DT @RT(15)tsRequiredPumps @RT(0) @T @T @UNKNOWN 0 @F
@F @F
@T
@BEG_Attrib
3 @RT(0) @RT(0) @RT(0)
@END_Attrib
1 0 @F @F @F @F

@Var @RT(18)sv_iDeviceForCalib @RT(0) @T @F @DT @RT(4)DINT @RT(0) @T @T @BASIC 0 @F
@F @F
@T
@BEG_Attrib
3 @RT(0) @RT(0) @RT(0)
@END_Attrib
1 8 @F @F @F @F

@Var @RT(15)mDeviceForCalib @RT(0) @T @T @DERIVED 0 @T @T @DT @RT(10)tsDeviceId @RT(0) @T @T @UNKNOWN 0 @F
@F @F
@T
@BEG_Attrib
3 @RT(0) @RT(0) @RT(0)
@END_Attrib
1 0 @F @F @F @F

@Var @RT(19)sv_PumpCalibDevices @RT(0) @T @T @DERIVED 0 @T @T @DT @RT(14)tyCalibDevices @RT(0) @T @T @UNKNOWN 0 @F
@F @F
@T
@BEG_Attrib
3 @RT(0) @RT(30)!!! device 1 - 20 reserved !!! @RT(0)
@END_Attrib
1 8 @F @F @F @F

@END_Dcl

@END_Export

@BEG_Body

6

@BEG_Export

@BEG_Algo
@POSTUPDATE_ALGORITHM @RT(6)pStart @STRUCTURED_TEXT
@RT(0) @RT(32)sv_CalibStatePumpPressure.Status @RT(9)PU_Task_7 @F @F
@END_Algo

@BEG_Dcl
@RT(16)DclTreeContainer
0
@END_Dcl

@END_Export

@BEG_Export

@BEG_Algo
@PROCESS_ALGORITHM @RT(5)paRun @SEQUENTIAL_FLOW_CHART
@RT(0) @RT(0) @RT(7)TaskMid @F @F
@END_Algo

@BEG_Dcl
@RT(16)DclTreeContainer
13
@Var @RT(7)uTmpCnt @RT(0) @T @F @DT @RT(5)UDINT @RT(0) @T @T @BASIC 0 @F
@F @F
@T
@BEG_Attrib
3 @RT(0) @RT(0) @RT(0)
@END_Attrib
1 4 @F @F @F @F

@Var @RT(18)evStartRequestData @RT(0) @T @T @DERIVED 0 @T @T @DT @RT(19)tevStartRequestData @RT(0) @T @T @UNKNOWN 0 @F
@F @F
@T
@BEG_Attrib
3 @RT(0) @RT(0) @RT(0)
@END_Attrib
1 0 @F @F @F @F

@Var @RT(12)fbCheckReady @RT(0) @T @T @DERIVED 0 @T @T @DT @RT(12)FBCheckReady @RT(0) @T @T @UNKNOWN 0 @F
@F @F
@T
@BEG_Attrib
3 @RT(0) @RT(0) @RT(0)
@END_Attrib
1 0 @F @F @F @F

@Var @RT(22)fbStopStartedMovements @RT(0) @T @T @DERIVED 0 @T @T @DT @RT(22)FBStopStartedMovements @RT(0) @T @T @UNKNOWN 0 @F
@F @F
@T
@BEG_Attrib
3 @RT(0) @RT(0) @RT(0)
@END_Attrib
1 0 @F @F @F @F

@Var @RT(5)fbLog @RT(0) @T @T @DERIVED 0 @T @T @DT @RT(14)FBAutoCalibLog @RT(0) @T @T @UNKNOWN 0 @F
@F @F
@T
@BEG_Attrib
3 @RT(0) @RT(0) @RT(0)
@END_Attrib
1 0 @F @F @F @F

@Var @RT(18)rMaxDetectPressure @RT(0) @T @F @DT @RT(4)REAL @RT(0) @T @T @BASIC 0 @F
@F @F
@T
@BEG_Attrib
3 @RT(0) @RT(27)Maximal identified pressure @RT(0)
@END_Attrib
1 0 @F @F @F @F

@Var @RT(7)rMinFac @RT(0) @T @F @DT @RT(4)REAL @RT(0) @T @T @BASIC 0 @F
@F @F
@T
@BEG_Attrib
3 @RT(4)0.05 @RT(78)security factor for checking difference of detected pressure and max. pressure @RT(0)
@END_Attrib
1 0 @F @F @F @F

@Var @RT(10)DelayTimer @RT(0) @T @T @DERIVED 0 @T @T @DT @RT(3)TON @RT(0) @T @T @UNKNOWN 0 @F
@F @F
@T
@BEG_Attrib
3 @RT(0) @RT(0) @RT(0)
@END_Attrib
1 0 @F @F @F @F

@Var @RT(22)OriginalPumpAssignment @RT(0) @T @T @DERIVED 0 @T @T @DT @RT(15)tyRequiredPumps @RT(0) @T @T @UNKNOWN 0 @F
@F @F
@T
@BEG_Attrib
3 @RT(0) @RT(0) @RT(0)
@END_Attrib
1 0 @F @F @F @F

@Var @RT(15)NoAssignedPumps @RT(0) @T @T @DERIVED 0 @T @T @DT @RT(15)tyRequiredPumps @RT(0) @T @T @UNKNOWN 0 @F
@F @F
@T
@BEG_Attrib
3 @RT(0) @RT(0) @RT(0)
@END_Attrib
1 0 @F @F @F @F

@Var @RT(13)tmpAssignment @RT(0) @T @T @DERIVED 0 @T @T @DT @RT(15)tyRequiredPumps @RT(0) @T @T @UNKNOWN 0 @F
@F @F
@T
@BEG_Attrib
3 @RT(0) @RT(0) @RT(0)
@END_Attrib
1 0 @F @F @F @F

@Var @RT(12)rMaxPressure @RT(0) @T @F @DT @RT(4)REAL @RT(0) @T @T @BASIC 0 @F
@F @F
@T
@BEG_Attrib
3 @RT(0) @RT(0) @RT(0)
@END_Attrib
1 0 @F @F @F @F

@Var @RT(20)abCreateMeasureArray @RT(0) @T @T @DERIVED 0 @T @T @DT @RT(20)ABCreateMeasureArray @RT(0) @T @T @UNKNOWN 0 @F
@F @F
@T
@BEG_Attrib
3 @RT(0) @RT(0) @RT(0)
@END_Attrib
1 0 @F @F @F @F

@END_Dcl

@END_Export

@BEG_Export

@BEG_Algo
@PROCESS_ALGORITHM @RT(16)paDeleteLogFiles @STRUCTURED_TEXT
@RT(0) @RT(0) @RT(8)TaskSlow @F @F
@END_Algo

@BEG_Dcl
@RT(16)DclTreeContainer
0
@END_Dcl

@END_Export

@BEG_Export

@BEG_Algo
@PROCESS_ALGORITHM @RT(14)paWriteLogFile @STRUCTURED_TEXT
@RT(0) @RT(0) @RT(8)TaskSlow @F @F
@END_Algo

@BEG_Dcl
@RT(16)DclTreeContainer
0
@END_Dcl

@END_Export

@BEG_Export

@BEG_Algo
@POSTUPDATE_ALGORITHM @RT(15)pPumpCalibError @STRUCTURED_TEXT
@RT(0) @RT(14)mpbCalibError^ @RT(9)PU_Task_7 @F @F
@END_Algo

@BEG_Dcl
@RT(16)DclTreeContainer
0
@END_Dcl

@END_Export

@BEG_Export

@BEG_Algo
@POSTUPDATE_ALGORITHM @RT(5)pInit @STRUCTURED_TEXT
@RT(0) @RT(31)sv_bInitDone,sv_iDeviceForCalib @RT(10)PU_Task_13 @F @F
@END_Algo

@BEG_Dcl
@RT(16)DclTreeContainer
0
@END_Dcl

@END_Export

@BEG_Body
@TL(20)
(**************************************** WARNING ********************************************
 *** The KEBA Kemro K2 System including software is not intended for safety control tasks! ***
 ***                       For further information see Comment tab!                        ***
 *********************************************************************************************)

IF sv_OperationMode = nSetup THEN
   IF sv_CalibStatePumpPressure.Status = tnCalibState_Running THEN
      IF sv_CalibStatePumpPressure.Group = tnCalibGroup_LintabOnly THEN
         //do not start pump calibration and set calib state to "done"
         sv_CalibStatePumpPressure.Status := tnCalibState_Done;
      ELSE
         sv_PumpCalibError.bError := FALSE;
         sv_PumpCalibError.iErrorInfo := 0;
         mpbCalibError := @sv_PumpCalibError.bError;
         START_PROCESS_ALGORITHM(paRun);
      END_IF;
   END_IF;
END_IF;

@END_Body

@@@BEG_Comment@@@
@TL(0)

@@@END_Comment@@@

@BEG_SfcBody
28 17 18

@BEG_SfcData 2
@StepSeq @RT(4)sseq @F 13
@Step @RT(7)S_RESET @F @F @T @F @RT(0) @F
@AcbCont @RT(7)unnamed @F 3
@Acb @RT(14)AStopmovements @F @F @RT(1)P @RT(0) @F @F @F @F
@Acb @RT(8)Action24 @F @T @RT(1)P @RT(0) @F @F @T @TL(7)
IF sv_CalibStatePumpPressure.Status <> tnCalibState_Error THEN
   fbLog('pressure calib aborted');
   sv_CalibStatePumpPressure.Status := tnCalibState_Aborted;
ELSE
   fbLog('pressure calib failure');
END_IF;

@F
@Acb @RT(10)AWaitReady @F @T @RT(1)N @RT(0) @F @F @T @TL(2)
fbCheckReady(DeviceId := mDeviceForCalib);

@F

@Trans @RT(17)TCalibDeviceReady @F @T @F @F @T @T @TL(2)
fbCheckReady.bReady AND mbLogFileSaved

@RT(7)Trans15 @F
@Step @RT(6)S_STOP @F @F @T @F @RT(0) @F
@AcbCont @RT(7)unnamed @F 1
@Acb @RT(8)Action22 @F @T @RT(1)P @RT(0) @F @F @T @TL(11)
sv_bDoPumpPressureCalib := FALSE;
mpbCalibError := EMPTY;
sv_iCalibratingPump := 0;
//restore original assignment
mpRequiredPumps^.RequiredPumps := OriginalPumpAssignment;

//delete dynamic arrays
abCreateMeasureArray.aRelease();

STOP_PROCESS_ALGORITHM();

@F

@Trans @RT(7)Trans18 @F @T @F @F @T @T @TL(2)
TRUE

@RT(7)Trans18 @F
@Step @RT(6)S_INIT @F @T @F @F @RT(0) @F
@AcbCont @RT(7)unnamed @F 2
@Acb @RT(5)AInit @F @T @RT(1)P @RT(0) @F @F @T @TL(10)
sv_bDoPumpPressureCalib := TRUE;
sv_bPumpPreVelCalibAnotherStepN := FALSE;
sv_bPumpPreVelCalibDone := FALSE;
sv_iCalibratingPump := sv_DeviceId.IndexId;
sv_CalibStatePumpPressure.prGlobalMaxX^ := sv_PumpData[sv_DeviceId.IndexId].prMaxPressure^;
sv_CalibStatePumpPressure.prGlobalMaxY^ := 10.0; //V

abCreateMeasureArray.aInit();  //create dynamic arrays
fbLog('pressure calib started');

@F
@Acb @RT(15)APumpAssignment @F @T @RT(1)P @RT(0) @F @F @T @TL(8)
//save actual pump assigment
OriginalPumpAssignment := mpRequiredPumps^.RequiredPumps;

//change assignment to the pump which should be calibrated
tmpAssignment := NoAssignedPumps;
tmpAssignment[sv_iCalibratingPump] := TRUE;
mpRequiredPumps^.RequiredPumps := tmpAssignment;

@F

@AltBranch @RT(3)alt @F 2
@TransSeq @RT(4)tseq @F 3
@Trans @RT(6)Trans1 @F @T @F @F @T @T @TL(3)
sv_TraceLevel.bDebugCalibration

@RT(6)Trans1 @F
@Step @RT(6)Step10 @F @F @F @F @RT(0) @F
@AcbCont @RT(7)unnamed @F 1
@Acb @RT(15)Delete_LogFiles @F @F @RT(1)P @RT(0) @F @F @T @F

@Trans @RT(7)Trans10 @F @T @F @F @T @T @TL(2)
mbFilesDeleted

@RT(7)Trans10 @F

@TransSeq @RT(4)tseq @F 1
@Trans @RT(7)Trans13 @F @T @T @F @T @T @TL(2)
NOT sv_TraceLevel.bDebugCalibration

@RT(7)Trans13 @F

@Step @RT(10)S_StartPos @F @F @F @F @RT(0) @F
@AcbCont @RT(7)unnamed @F 2
@Acb @RT(13)AMoveStartPos @F @F @RT(1)P @RT(0) @F @F @F @F
@Acb @RT(7)Action8 @F @T @RT(1)N @RT(0) @F @F @T @TL(2)
fbCheckReady(DeviceId := mDeviceForCalib);

@F

@Trans @RT(6)Trans5 @F @T @F @F @T @T @TL(2)
fbCheckReady.bReady

@RT(6)Trans5 @F
@Loop @RT(4)loop @F 2
@StepSeq @RT(4)sseq @F 5
@Step @RT(7)S_Calib @F @F @F @F @RT(0) @F
@AcbCont @RT(7)unnamed @F 2
@Acb @RT(6)ACalib @F @F @RT(1)P @RT(0) @F @F @F @F
@Acb @RT(7)Action9 @F @T @RT(1)N @RT(0) @F @F @T @TL(2)
fbCheckReady(DeviceId := mDeviceForCalib);

@F

@Trans @RT(6)Trans2 @F @T @F @F @T @T @TL(2)
fbCheckReady.bReady

@RT(6)Trans2 @F
@Step @RT(11)S_WAIT_CALC @F @F @F @F @RT(0) @F
@AcbCont @RT(7)unnamed @F 1
@Acb @RT(8)Action27 @F @T @RT(1)P @RT(0) @F @F @T @TL(10)
//show lintab during calibration
sv_CalibStatePumpPressure.pDisplayLintab^.LintabPoints.uNoOfPoints := sv_TmpLintab.LintabPoints.uNoOfPoints;
FOR uTmpCnt := 1 TO sv_TmpLintab.LintabPoints.uNoOfPoints DO
   sv_CalibStatePumpPressure.pDisplayLintab^.LintabPoints.Point[uTmpCnt].rX:= sv_TmpLintab.LintabPoints.Point[uTmpCnt].rX;
   sv_CalibStatePumpPressure.pDisplayLintab^.LintabPoints.Point[uTmpCnt].rY:= sv_TmpLintab.LintabPoints.Point[uTmpCnt].rY;
END_FOR;
DelayTimer(IN:=FALSE);
DelayTimer(IN:=TRUE, PT:=sv_dDelayTimeNextShot);

@F

@AltBranch @RT(3)alt @F 2
@TransSeq @RT(4)tseq @F 3
@Trans @RT(7)Trans14 @F @T @F @F @T @T @TL(2)
sv_TraceLevel.bDebugCalibration

@RT(7)Trans14 @F
@Step @RT(6)Step11 @F @F @F @F @RT(0) @F
@AcbCont @RT(7)unnamed @F 1
@Acb @RT(13)Write_LogFile @F @F @RT(1)P @RT(0) @F @F @T @F

@Trans @RT(7)Trans30 @F @T @F @F @T @T @TL(2)
mbLogFileSaved

@RT(7)Trans15 @F

@TransSeq @RT(4)tseq @F 1
@Trans @RT(7)Trans16 @F @T @T @F @T @T @TL(2)
NOT sv_TraceLevel.bDebugCalibration

@RT(7)Trans16 @F

@Step @RT(6)Step12 @F @F @F @F @RT(0) @F
@AcbCont @RT(7)unnamed @F 1
@Acb @RT(9)WaitDelay @F @T @RT(1)N @RT(0) @F @F @T @TL(2)
DelayTimer(IN:=TRUE);

@F

@Trans @RT(7)Trans24 @F @T @T @T @T @T @TL(4)
sv_bPumpPreVelCalibAnotherStepN AND
DelayTimer.Q
// another step needed

@RT(7)Trans24 @F

@AltBranch @RT(3)alt @F 2
@TransSeq @RT(4)tseq @F 1
@Trans @RT(7)Trans21 @F @T @F @F @T @T @TL(3)
sv_bPumpPreVelCalibDone
//calib finished

@RT(7)Trans21 @F

@TransSeq @RT(4)tseq @F 2
@Trans @RT(7)Trans23 @F @T @F @F @T @T @TL(4)
NOT sv_bPumpPreVelCalibAnotherStepN
AND NOT sv_bPumpPreVelCalibDone
//maybe remove in vlavour of exit

@RT(7)Trans23 @F
@Goto @RT(7)S_RESET @F @F

@Step @RT(6)S_DONE @F @F @F @F @RT(0) @F
@AcbCont @RT(7)unnamed @F 2
@Acb @RT(8)Action18 @F @T @RT(1)P @RT(0) @F @F @T @TL(5)
//copy lintab and set calib state
fbLog('pressure calib finished');
sv_PressureLintab := sv_CalibStatePumpPressure.pDisplayLintab^;
sv_CalibStatePumpPressure.Status := tnCalibState_Done;

@F
@Acb @RT(21)ACompareToMaxPressure @F @F @RT(1)P @RT(0) @F @F @F @F

@Trans @RT(7)Trans19 @F @T @F @F @T @T @TL(2)
TRUE

@RT(7)Trans19 @F
@Goto @RT(6)S_STOP @F @F
@END_SfcData
@SaActions 6
@SaText @RT(13)AMoveStartPos 1 @TL(10)
(**************************************** WARNING ********************************************
 *** The KEBA Kemro K2 System including software is not intended for safety control tasks! ***
 ***                       For further information see Comment tab!                        ***
 *********************************************************************************************)

evStartRequestData.DeviceId := mDeviceForCalib;
evStartRequestData.MoveDir := mMoveDirStartPos;
evStartRequestData.MoveId := mMoveIdStartPos;
SET_EVENT(evStartRequest, evStartRequestData);

@SaText @RT(14)AStopmovements 1 @TL(7)
(**************************************** WARNING ********************************************
 *** The KEBA Kemro K2 System including software is not intended for safety control tasks! ***
 ***                       For further information see Comment tab!                        ***
 *********************************************************************************************)

fbStopStartedMovements();

@SaText @RT(6)ACalib 1 @TL(10)
(**************************************** WARNING ********************************************
 *** The KEBA Kemro K2 System including software is not intended for safety control tasks! ***
 ***                       For further information see Comment tab!                        ***
 *********************************************************************************************)

evStartRequestData.DeviceId := mDeviceForCalib;
evStartRequestData.MoveDir := mMoveDirCalib;
evStartRequestData.MoveId := mMoveIdCalib;
SET_EVENT(evStartRequest, evStartRequestData);

@SaText @RT(21)ACompareToMaxPressure 1 @TL(14)
(**************************************** WARNING ********************************************
 *** The KEBA Kemro K2 System including software is not intended for safety control tasks! ***
 ***                       For further information see Comment tab!                        ***
 *********************************************************************************************)

// Set alarm if detected pressure differs too strong from max. pressure
rMaxDetectPressure := sv_PressureLintab.LintabPoints.Point[sv_PressureLintab.LintabPoints.uNoOfPoints].rX;
rMaxPressure := sv_PumpData[sv_DeviceId.IndexId].prMaxPressure^;
IF ABS(rMaxPressure - rMaxDetectPressure) > (rMinFac * rMaxPressure) THEN
   SET_ALARM(Name := erHighDiffAtPres,
             SubID1 := sv_DeviceId.CompId,
             SubID2 := sv_DeviceId.IndexId);
END_IF;

@SaText @RT(15)Delete_LogFiles 1 @TL(9)
(**************************************** WARNING ********************************************
 *** The KEBA Kemro K2 System including software is not intended for safety control tasks! ***
 ***                       For further information see Comment tab!                        ***
 *********************************************************************************************)

mbFilesDeleted := FALSE;
START_PROCESS_ALGORITHM(paDeleteLogFiles);

@SaText @RT(13)Write_LogFile 1 @TL(8)
(**************************************** WARNING ********************************************
 *** The KEBA Kemro K2 System including software is not intended for safety control tasks! ***
 ***                       For further information see Comment tab!                        ***
 *********************************************************************************************)

mbLogFileSaved := FALSE;
START_PROCESS_ALGORITHM(paWriteLogFile);

@SaTrans 0
@SaExits 2
@SaExit @SaText @RT(14)E_NotSetupMode 1 @TL(7)
(**************************************** WARNING ********************************************
 *** The KEBA Kemro K2 System including software is not intended for safety control tasks! ***
 ***                       For further information see Comment tab!                        ***
 *********************************************************************************************)

sv_OperationMode <> nSetup

@RT(7)S_RESET @RT(1)1 @F @F @SaSfc @RT(14)E_NotSetupMode 5 @RT(5)DUMMY
@BEG_SfcData 2
@ExitSeq @RT(4)sseq @F 3
@Step @RT(8)unnamed1 @F @T @F @F @RT(0) @F
@AcbCont @RT(7)unnamed @F 0

@Trans @RT(8)unnamed3 @F @T @F @F @T @T @TL(2)

@RT(8)unnamed3 @F
@Goto @RT(9)unlabeled @F @F
@END_SfcData

@SaExit @SaText @RT(23)E_NotCalibratingAnymore 1 @TL(3)
// abort calibration, when not in running state and not finished
sv_CalibStatePumpPressure.Status <> tnCalibState_Running AND (S_INIT.X OR S_StartPos.X OR S_Calib.X OR S_WAIT_CALC.X)

@RT(7)S_RESET @RT(1)1 @F @F @SaSfc @RT(23)E_NotCalibratingAnymore 5 @RT(5)DUMMY
@BEG_SfcData 2
@ExitSeq @RT(4)sseq @F 3
@Step @RT(8)unnamed4 @F @T @F @F @RT(0) @F
@AcbCont @RT(7)unnamed @F 0

@Trans @RT(8)unnamed6 @F @T @F @F @T @T @TL(2)

@RT(8)unnamed6 @F
@Goto @RT(9)unlabeled @F @F
@END_SfcData

@END_SfcBody

@@@BEG_Comment@@@
@TL(0)

@@@END_Comment@@@

@BEG_Body
@TL(9)
(**************************************** WARNING ********************************************
 *** The KEBA Kemro K2 System including software is not intended for safety control tasks! ***
 ***                       For further information see Comment tab!                        ***
 *********************************************************************************************)

fbCalibWriteLog(fileName:=cCalibFilePres,bDeleteFiles:=TRUE);
mbFilesDeleted := TRUE;
STOP_PROCESS_ALGORITHM();

@END_Body

@@@BEG_Comment@@@
@TL(0)

@@@END_Comment@@@

@BEG_Body
@TL(9)
(**************************************** WARNING ********************************************
 *** The KEBA Kemro K2 System including software is not intended for safety control tasks! ***
 ***                       For further information see Comment tab!                        ***
 *********************************************************************************************)

fbCalibWriteLog(fileName:= cCalibFilePres,bDeleteFiles := FALSE);
mbLogFileSaved := TRUE;
STOP_PROCESS_ALGORITHM();

@END_Body

@@@BEG_Comment@@@
@TL(0)

@@@END_Comment@@@

@BEG_Body
@TL(16)
(**************************************** WARNING ********************************************
 *** The KEBA Kemro K2 System including software is not intended for safety control tasks! ***
 ***                       For further information see Comment tab!                        ***
 *********************************************************************************************)

IF sv_PumpCalibError.bError THEN

   sv_CalibStatePumpPressure.Status := tnCalibState_Error;
   IF sv_PumpCalibError.iErrorInfo = cValueChangeDuringCalibTooLow THEN
      SET_ALARM(erPumpPresCalibNoValueChange);
   ELSE
      SET_ALARM(erCalibrationPressureNotStable);
   END_IF;

END_IF;

@END_Body

@@@BEG_Comment@@@
@TL(0)

@@@END_Comment@@@

@BEG_Body
@TL(35)
(**************************************** WARNING ********************************************
 *** The KEBA Kemro K2 System including software is not intended for safety control tasks! ***
 ***                       For further information see Comment tab!                        ***
 *********************************************************************************************)

mDeviceForCalib.CompId := cMinCompId;
mDeviceForCalib.IndexId := cMinMoveIdent;
mMoveDirStartPos := cMinMoveIdent;
mMoveIdStartPos := cMinMoveIdent;
mMoveDirCalib := cMinMoveIdent;
mMoveIdCalib := cMinMoveIdent;
mpRequiredPumps := EMPTY;
sv_CalibStatePumpPressure.prInputSensor := EMPTY;
sv_CalibStatePumpPressure.Group := tnCalibGroup_LintabOnly;

IF (sv_iDeviceForCalib > 0) AND (sv_iDeviceForCalib <= cMaxCalibDevices) THEN
   mDeviceForCalib := sv_PumpCalibDevices[sv_iDeviceForCalib].DeviceId;

   IF CHECK_REF(sv_PumpCalibDevices[sv_iDeviceForCalib].pPresCalibStartPosMovement^) THEN
      mMoveDirStartPos := sv_PumpCalibDevices[sv_iDeviceForCalib].pPresCalibStartPosMovement^.MoveDir;
      mMoveIdStartPos :=  sv_PumpCalibDevices[sv_iDeviceForCalib].pPresCalibStartPosMovement^.MoveId;
   END_IF;

   IF CHECK_REF(sv_PumpCalibDevices[sv_iDeviceForCalib].pPresCalibMovement^) THEN
      mMoveDirCalib := sv_PumpCalibDevices[sv_iDeviceForCalib].pPresCalibMovement^.MoveDir;
      mMoveIdCalib := sv_PumpCalibDevices[sv_iDeviceForCalib].pPresCalibMovement^.MoveId;
      mpRequiredPumps := sv_PumpCalibDevices[sv_iDeviceForCalib].pPresCalibMovement^.AnaOutData.pRequiredPumps;
   END_IF;

   IF CHECK_REF(sv_PumpCalibDevices[sv_iDeviceForCalib].prActPressure^) THEN
      sv_CalibStatePumpPressure.prInputSensor := sv_PumpCalibDevices[sv_iDeviceForCalib].prActPressure;
      sv_CalibStatePumpPressure.Group := tnCalibGroup_Pressure;
   END_IF;
END_IF;

@END_Body

@@@BEG_Comment@@@
@TL(0)

@@@END_Comment@@@
@END_Body

@END_Contents
